Yaskawa INFORM job: A_ROOF_SIDE_0617_2_PAINT_0.JBI

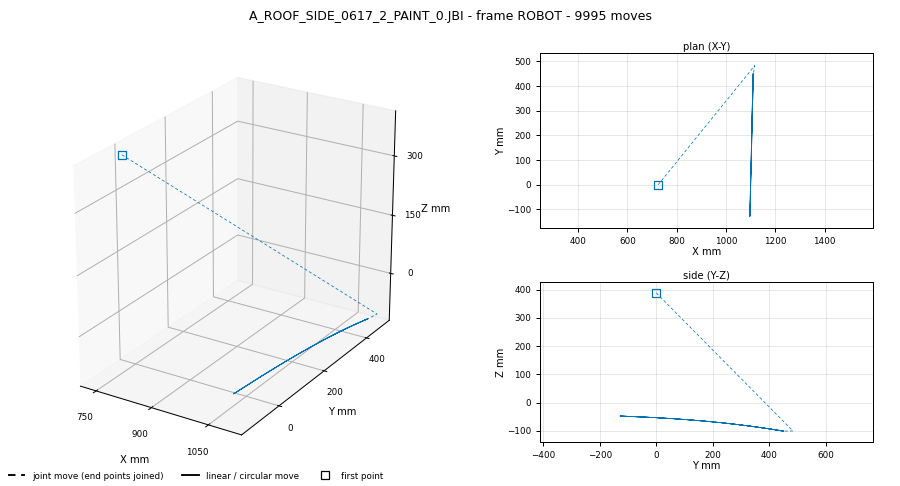
[picture p0: tool path of A_ROOF_SIDE_0617_2_PAINT_0.JBI in frame ROBOT, 9995 of 9995 moves have a stored position in this frame; points joined in program order, loops and branches not executed]
/JOB
//NAME A_ROOF_SIDE_0617_2_PAINT
//POS
///NPOS 9995,0,0,0,0,0
///TOOL 0
///USER 0
///POSTYPE ROBOT
///RECTAN
///RCONF 1,0,0,0,0,0,0,0,0,0,0,0,0,0,0,0,0,0,0,0,0,0,0,0
C00000=725.000,0.000,388.500,-180.000,-0.000,0.000
C00001=725.000,0.000,388.500,-180.000,-0.000,0.000
///TOOL 1
///USER 0
///POSTYPE ROBOT
///RECTAN
C00002=1116.924,483.635,-100.044,-178.124,16.519,151.125
C00003=1111.077,450.492,-100.420,-178.124,16.519,151.125
C00004=1111.072,450.245,-100.379,-178.121,16.509,151.122
C00005=1111.067,450.000,-100.338,-178.120,16.499,151.119
C00006=1111.061,449.753,-100.297,-178.118,16.490,151.116
C00007=1111.056,449.506,-100.255,-178.115,16.481,151.114
C00008=1111.050,449.260,-100.213,-178.113,16.472,151.111
C00009=1111.045,449.013,-100.173,-178.111,16.462,151.108
C00010=1111.039,448.767,-100.131,-178.109,16.453,151.105
C00011=1111.034,448.521,-100.090,-178.107,16.443,151.102
C00012=1111.028,448.275,-100.049,-178.105,16.434,151.099
C00013=1111.023,448.027,-100.007,-178.103,16.424,151.096
C00014=1111.017,447.781,-99.966,-178.102,16.415,151.094
C00015=1111.012,447.534,-99.925,-178.100,16.405,151.091
C00016=1111.007,447.289,-99.884,-178.099,16.395,151.088
C00017=1111.002,447.042,-99.843,-178.098,16.386,151.085
C00018=1110.996,446.796,-99.801,-178.096,16.376,151.082
C00019=1110.991,446.548,-99.760,-178.095,16.367,151.080
C00020=1110.985,446.302,-99.719,-178.093,16.357,151.077
C00021=1110.980,446.056,-99.678,-178.092,16.348,151.074
C00022=1110.975,445.810,-99.636,-178.092,16.338,151.072
C00023=1110.969,445.563,-99.595,-178.091,16.328,151.069
C00024=1110.963,445.317,-99.554,-178.090,16.318,151.066
C00025=1110.957,445.070,-99.513,-178.089,16.309,151.064
C00026=1110.952,444.824,-99.473,-178.089,16.299,151.061
C00027=1110.947,444.577,-99.431,-178.088,16.290,151.058
C00028=1110.941,444.330,-99.390,-178.088,16.280,151.056
C00029=1110.935,444.084,-99.349,-178.088,16.270,151.053
C00030=1110.930,443.838,-99.308,-178.088,16.260,151.051
C00031=1110.925,443.591,-99.267,-178.087,16.251,151.048
C00032=1110.919,443.345,-99.226,-178.087,16.241,151.046
C00033=1110.915,443.099,-99.185,-178.088,16.231,151.043
C00034=1110.909,442.852,-99.144,-178.088,16.221,151.041
C00035=1110.903,442.605,-99.103,-178.088,16.212,151.038
C00036=1110.898,442.359,-99.062,-178.089,16.202,151.036
C00037=1110.892,442.113,-99.022,-178.088,16.192,151.033
C00038=1110.887,441.866,-98.981,-178.089,16.182,151.031
C00039=1110.881,441.620,-98.940,-178.089,16.173,151.028
C00040=1110.876,441.373,-98.899,-178.089,16.164,151.026
C00041=1110.870,441.127,-98.858,-178.090,16.154,151.024
C00042=1110.864,440.880,-98.818,-178.090,16.145,151.021
C00043=1110.859,440.634,-98.777,-178.090,16.136,151.019
C00044=1110.853,440.387,-98.736,-178.091,16.126,151.017
C00045=1110.848,440.141,-98.695,-178.092,16.117,151.014
C00046=1110.843,439.894,-98.655,-178.092,16.107,151.012
C00047=1110.837,439.648,-98.614,-178.093,16.098,151.010
C00048=1110.831,439.401,-98.573,-178.093,16.089,151.007
C00049=1110.826,439.155,-98.533,-178.093,16.080,151.005
C00050=1110.820,438.908,-98.493,-178.094,16.071,151.003
C00051=1110.814,438.661,-98.452,-178.095,16.061,151.001
C00052=1110.809,438.428,-98.413,-178.095,16.052,150.998
C00053=1110.804,438.194,-98.375,-178.095,16.044,150.996
C00054=1110.799,437.961,-98.337,-178.096,16.036,150.994
C00055=1110.794,437.728,-98.298,-178.096,16.027,150.992
C00056=1110.788,437.494,-98.260,-178.097,16.019,150.990
C00057=1110.783,437.261,-98.221,-178.098,16.010,150.988
C00058=1110.778,437.027,-98.183,-178.098,16.002,150.986
C00059=1110.773,436.795,-98.145,-178.099,15.993,150.984
C00060=1110.767,436.548,-98.105,-178.100,15.985,150.982
C00061=1110.761,436.301,-98.064,-178.100,15.976,150.980
C00062=1110.756,436.055,-98.023,-178.101,15.967,150.978
C00063=1110.751,435.808,-97.983,-178.102,15.958,150.976
C00064=1110.745,435.562,-97.944,-178.103,15.949,150.973
C00065=1110.740,435.315,-97.903,-178.103,15.941,150.971
C00066=1110.734,435.068,-97.862,-178.104,15.932,150.969
C00067=1110.729,434.822,-97.822,-178.104,15.924,150.967
C00068=1110.723,434.575,-97.782,-178.105,15.915,150.965
C00069=1110.718,434.329,-97.742,-178.106,15.906,150.963
C00070=1110.712,434.082,-97.701,-178.107,15.898,150.961
C00071=1110.707,433.836,-97.661,-178.108,15.889,150.959
C00072=1110.701,433.589,-97.621,-178.109,15.881,150.957
C00073=1110.696,433.343,-97.581,-178.110,15.872,150.955
C00074=1110.690,433.096,-97.540,-178.111,15.864,150.953
C00075=1110.684,432.849,-97.501,-178.111,15.856,150.951
C00076=1110.679,432.602,-97.460,-178.112,15.847,150.949
C00077=1110.674,432.356,-97.420,-178.113,15.839,150.947
C00078=1110.668,432.109,-97.381,-178.114,15.831,150.945
C00079=1110.662,431.862,-97.340,-178.115,15.823,150.943
C00080=1110.657,431.616,-97.301,-178.116,15.815,150.942
C00081=1110.651,431.369,-97.260,-178.117,15.807,150.940
C00082=1110.646,431.123,-97.220,-178.118,15.798,150.938
C00083=1110.640,430.876,-97.180,-178.119,15.790,150.936
C00084=1110.635,430.630,-97.140,-178.120,15.782,150.934
C00085=1110.629,430.383,-97.100,-178.121,15.774,150.932
C00086=1110.623,430.136,-97.060,-178.122,15.766,150.930
C00087=1110.618,429.889,-97.021,-178.123,15.758,150.928
C00088=1110.612,429.642,-96.980,-178.124,15.750,150.927
C00089=1110.607,429.396,-96.941,-178.125,15.742,150.925
C00090=1110.602,429.149,-96.901,-178.126,15.734,150.923
C00091=1110.596,428.903,-96.861,-178.127,15.726,150.921
C00092=1110.590,428.655,-96.821,-178.128,15.719,150.919
C00093=1110.585,428.410,-96.781,-178.130,15.711,150.918
C00094=1110.579,428.162,-96.742,-178.131,15.703,150.916
C00095=1110.574,427.916,-96.702,-178.132,15.695,150.914
C00096=1110.567,427.669,-96.662,-178.133,15.687,150.912
C00097=1110.563,427.422,-96.622,-178.134,15.680,150.911
C00098=1110.557,427.175,-96.583,-178.135,15.672,150.909
C00099=1110.551,426.929,-96.544,-178.136,15.665,150.907
C00100=1110.546,426.682,-96.503,-178.138,15.657,150.906
C00101=1110.540,426.436,-96.464,-178.139,15.649,150.904
C00102=1110.534,426.188,-96.425,-178.140,15.642,150.902
C00103=1110.529,425.942,-96.385,-178.141,15.635,150.901
C00104=1110.523,425.696,-96.345,-178.142,15.627,150.899
C00105=1110.518,425.448,-96.305,-178.144,15.620,150.897
C00106=1110.513,425.202,-96.266,-178.145,15.612,150.896
C00107=1110.507,424.955,-96.227,-178.146,15.604,150.894
C00108=1110.502,424.737,-96.191,-178.148,15.598,150.893
C00109=1110.497,424.520,-96.157,-178.149,15.591,150.891
C00110=1110.492,424.301,-96.122,-178.150,15.585,150.890
C00111=1110.487,424.083,-96.087,-178.151,15.579,150.888
C00112=1110.483,423.866,-96.052,-178.152,15.572,150.887
C00113=1110.477,423.649,-96.018,-178.153,15.566,150.885
C00114=1110.472,423.430,-95.983,-178.154,15.560,150.884
C00115=1110.468,423.213,-95.948,-178.155,15.553,150.883
C00116=1110.462,422.966,-95.909,-178.157,15.546,150.881
C00117=1110.456,422.719,-95.870,-178.158,15.538,150.880
C00118=1110.451,422.472,-95.830,-178.160,15.531,150.878
C00119=1110.446,422.226,-95.791,-178.161,15.524,150.877
C00120=1110.440,421.979,-95.752,-178.163,15.517,150.875
C00121=1110.434,421.732,-95.712,-178.164,15.510,150.874
C00122=1110.429,421.486,-95.673,-178.165,15.503,150.872
C00123=1110.422,421.238,-95.634,-178.167,15.496,150.871
C00124=1110.417,420.992,-95.595,-178.169,15.489,150.869
C00125=1110.412,420.745,-95.556,-178.170,15.483,150.868
C00126=1110.407,420.497,-95.516,-178.171,15.475,150.866
C00127=1110.401,420.251,-95.477,-178.173,15.468,150.865
C00128=1110.395,420.004,-95.438,-178.174,15.462,150.863
C00129=1110.389,419.757,-95.399,-178.176,15.455,150.862
C00130=1110.384,419.511,-95.360,-178.177,15.448,150.860
C00131=1110.378,419.263,-95.321,-178.179,15.441,150.859
C00132=1110.373,419.017,-95.282,-178.181,15.434,150.858
C00133=1110.367,418.770,-95.243,-178.182,15.428,150.856
C00134=1110.361,418.523,-95.203,-178.184,15.421,150.855
C00135=1110.356,418.276,-95.165,-178.185,15.415,150.854
C00136=1110.351,418.030,-95.126,-178.187,15.408,150.852
C00137=1110.345,417.783,-95.087,-178.188,15.401,150.851
C00138=1110.339,417.536,-95.048,-178.190,15.394,150.850
C00139=1110.334,417.289,-95.009,-178.191,15.388,150.848
C00140=1110.328,417.042,-94.970,-178.193,15.381,150.847
C00141=1110.323,416.795,-94.931,-178.194,15.375,150.845
C00142=1110.317,416.549,-94.892,-178.196,15.368,150.844
C00143=1110.311,416.301,-94.854,-178.197,15.362,150.843
C00144=1110.306,416.054,-94.814,-178.199,15.355,150.842
C00145=1110.301,415.807,-94.776,-178.201,15.349,150.840
C00146=1110.295,415.560,-94.737,-178.203,15.342,150.839
C00147=1110.288,415.314,-94.698,-178.204,15.336,150.838
C00148=1110.283,415.067,-94.660,-178.206,15.330,150.836
C00149=1110.277,414.820,-94.620,-178.208,15.323,150.835
C00150=1110.272,414.573,-94.582,-178.210,15.317,150.834
C00151=1110.267,414.326,-94.544,-178.211,15.311,150.833
C00152=1110.261,414.079,-94.505,-178.213,15.305,150.832
C00153=1110.255,413.832,-94.467,-178.215,15.298,150.830
C00154=1110.249,413.585,-94.427,-178.216,15.292,150.829
C00155=1110.244,413.338,-94.389,-178.218,15.286,150.828
C00156=1110.238,413.091,-94.350,-178.220,15.280,150.827
C00157=1110.232,412.844,-94.312,-178.222,15.274,150.826
C00158=1110.227,412.597,-94.274,-178.224,15.267,150.824
C00159=1110.222,412.351,-94.235,-178.225,15.261,150.823
C00160=1110.216,412.103,-94.196,-178.227,15.255,150.822
C00161=1110.211,411.856,-94.157,-178.229,15.249,150.821
C00162=1110.205,411.609,-94.120,-178.231,15.243,150.820
C00163=1110.199,411.363,-94.081,-178.232,15.237,150.818
C00164=1110.194,411.151,-94.048,-178.234,15.232,150.818
C00165=1110.190,410.939,-94.015,-178.235,15.227,150.817
C00166=1110.185,410.729,-93.982,-178.237,15.222,150.816
C00167=1110.180,410.517,-93.949,-178.238,15.217,150.815
C00168=1110.176,410.305,-93.917,-178.240,15.211,150.814
C00169=1110.171,410.094,-93.883,-178.241,15.207,150.813
C00170=1110.166,409.883,-93.851,-178.243,15.201,150.812
C00171=1110.161,409.671,-93.818,-178.244,15.197,150.811
C00172=1110.156,409.424,-93.780,-178.247,15.190,150.810
C00173=1110.150,409.177,-93.740,-178.248,15.185,150.809
C00174=1110.144,408.931,-93.703,-178.250,15.179,150.808
C00175=1110.139,408.683,-93.664,-178.252,15.173,150.806
C00176=1110.134,408.436,-93.626,-178.253,15.168,150.805
C00177=1110.128,408.190,-93.588,-178.256,15.161,150.804
C00178=1110.123,407.943,-93.550,-178.258,15.156,150.803
C00179=1110.116,407.695,-93.512,-178.259,15.150,150.802
C00180=1110.111,407.448,-93.473,-178.261,15.145,150.801
C00181=1110.105,407.201,-93.436,-178.263,15.139,150.800
C00182=1110.100,406.954,-93.397,-178.266,15.133,150.799
C00183=1110.095,406.707,-93.359,-178.267,15.127,150.798
C00184=1110.089,406.461,-93.321,-178.269,15.122,150.797
C00185=1110.084,406.213,-93.283,-178.271,15.116,150.796
C00186=1110.077,405.966,-93.245,-178.273,15.111,150.795
C00187=1110.072,405.719,-93.206,-178.275,15.105,150.794
C00188=1110.066,405.472,-93.169,-178.277,15.100,150.793
C00189=1110.061,405.225,-93.130,-178.279,15.095,150.792
C00190=1110.055,404.978,-93.093,-178.281,15.089,150.791
C00191=1110.049,404.731,-93.056,-178.283,15.084,150.791
C00192=1110.044,404.484,-93.017,-178.285,15.078,150.790
C00193=1110.038,404.237,-92.979,-178.287,15.073,150.789
C00194=1110.033,403.989,-92.941,-178.289,15.067,150.788
C00195=1110.027,403.743,-92.903,-178.291,15.062,150.787
C00196=1110.021,403.496,-92.865,-178.293,15.057,150.786
C00197=1110.016,403.248,-92.828,-178.295,15.051,150.785
C00198=1110.010,403.002,-92.790,-178.297,15.046,150.784
C00199=1110.004,402.755,-92.752,-178.299,15.041,150.783
C00200=1109.999,402.508,-92.714,-178.301,15.035,150.782
C00201=1109.993,402.260,-92.677,-178.303,15.030,150.781
C00202=1109.987,402.014,-92.639,-178.305,15.025,150.781
C00203=1109.982,401.767,-92.601,-178.307,15.020,150.780
C00204=1109.977,401.519,-92.563,-178.309,15.014,150.779
C00205=1109.971,401.273,-92.526,-178.312,15.009,150.778
C00206=1109.966,401.025,-92.487,-178.313,15.004,150.777
C00207=1109.960,400.778,-92.450,-178.316,14.999,150.776
C00208=1109.954,400.531,-92.413,-178.317,14.995,150.775
C00209=1109.949,400.284,-92.375,-178.319,14.989,150.775
C00210=1109.943,400.037,-92.337,-178.321,14.984,150.774
C00211=1109.937,399.790,-92.299,-178.324,14.979,150.773
C00212=1109.932,399.543,-92.262,-178.326,14.974,150.772
C00213=1109.926,399.296,-92.225,-178.328,14.969,150.771
C00214=1109.921,399.048,-92.187,-178.330,14.964,150.771
C00215=1109.915,398.801,-92.149,-178.332,14.959,150.770
C00216=1109.909,398.554,-92.112,-178.335,14.954,150.769
C00217=1109.904,398.308,-92.074,-178.337,14.949,150.768
C00218=1109.898,398.060,-92.037,-178.339,14.945,150.767
C00219=1109.892,397.813,-92.000,-178.341,14.940,150.767
C00220=1109.888,397.601,-91.967,-178.343,14.936,150.766
C00221=1109.883,397.390,-91.935,-178.345,14.931,150.765
C00222=1109.878,397.178,-91.904,-178.347,14.927,150.765
C00223=1109.873,396.966,-91.871,-178.349,14.923,150.764
C00224=1109.868,396.755,-91.839,-178.350,14.919,150.763
C00225=1109.863,396.543,-91.808,-178.352,14.915,150.763
C00226=1109.858,396.331,-91.775,-178.354,14.911,150.762
C00227=1109.854,396.119,-91.743,-178.356,14.907,150.762
C00228=1109.848,395.872,-91.706,-178.358,14.902,150.761
C00229=1109.842,395.625,-91.669,-178.360,14.897,150.760
C00230=1109.837,395.378,-91.632,-178.363,14.892,150.760
C00231=1109.831,395.132,-91.594,-178.365,14.887,150.759
C00232=1109.826,394.884,-91.557,-178.367,14.883,150.758
C00233=1109.820,394.637,-91.520,-178.369,14.878,150.757
C00234=1109.815,394.389,-91.483,-178.372,14.874,150.757
C00235=1109.809,394.143,-91.445,-178.374,14.869,150.756
C00236=1109.803,393.895,-91.408,-178.376,14.865,150.755
C00237=1109.797,393.648,-91.371,-178.379,14.860,150.755
C00238=1109.792,393.401,-91.334,-178.381,14.855,150.754
C00239=1109.787,393.155,-91.297,-178.383,14.850,150.753
C00240=1109.781,392.907,-91.260,-178.385,14.847,150.753
C00241=1109.775,392.660,-91.223,-178.387,14.842,150.752
C00242=1109.770,392.413,-91.186,-178.390,14.837,150.752
C00243=1109.764,392.165,-91.149,-178.393,14.832,150.751
C00244=1109.758,391.918,-91.112,-178.394,14.828,150.750
C00245=1109.752,391.671,-91.074,-178.397,14.824,150.750
C00246=1109.746,391.424,-91.037,-178.400,14.819,150.749
C00247=1109.741,391.177,-91.001,-178.401,14.815,150.749
C00248=1109.736,390.930,-90.964,-178.404,14.811,150.748
C00249=1109.729,390.683,-90.927,-178.407,14.806,150.748
C00250=1109.724,390.436,-90.890,-178.410,14.802,150.747
C00251=1109.718,390.188,-90.853,-178.411,14.798,150.746
C00252=1109.713,389.942,-90.816,-178.414,14.793,150.746
C00253=1109.707,389.694,-90.780,-178.417,14.788,150.745
C00254=1109.701,389.447,-90.743,-178.419,14.785,150.745
C00255=1109.696,389.200,-90.706,-178.421,14.780,150.744
C00256=1109.690,388.952,-90.669,-178.424,14.776,150.744
C00257=1109.684,388.706,-90.633,-178.426,14.772,150.743
C00258=1109.679,388.459,-90.596,-178.429,14.767,150.743
C00259=1109.673,388.211,-90.559,-178.432,14.763,150.742
C00260=1109.667,387.964,-90.522,-178.433,14.759,150.741
C00261=1109.662,387.718,-90.486,-178.436,14.755,150.741
C00262=1109.656,387.470,-90.449,-178.438,14.751,150.740
C00263=1109.650,387.223,-90.412,-178.441,14.747,150.740
C00264=1109.645,386.976,-90.376,-178.444,14.742,150.739
C00265=1109.640,386.729,-90.339,-178.446,14.738,150.739
C00266=1109.633,386.481,-90.303,-178.448,14.734,150.738
C00267=1109.628,386.234,-90.266,-178.451,14.729,150.738
C00268=1109.623,385.987,-90.229,-178.453,14.726,150.738
C00269=1109.617,385.740,-90.193,-178.456,14.721,150.737
C00270=1109.611,385.492,-90.156,-178.458,14.718,150.737
C00271=1109.606,385.246,-90.120,-178.461,14.713,150.736
C00272=1109.600,384.999,-90.083,-178.464,14.709,150.736
C00273=1109.594,384.751,-90.047,-178.466,14.706,150.735
C00274=1109.589,384.504,-90.011,-178.469,14.701,150.735
C00275=1109.583,384.257,-89.974,-178.471,14.697,150.734
C00276=1109.573,383.845,-89.913,-178.476,14.691,150.734
C00277=1109.564,383.434,-89.853,-178.479,14.684,150.733
C00278=1109.555,383.023,-89.792,-178.484,14.677,150.732
C00279=1109.546,382.612,-89.732,-178.488,14.671,150.732
C00280=1109.540,382.364,-89.695,-178.491,14.667,150.731
C00281=1109.534,382.117,-89.659,-178.493,14.663,150.731
C00282=1109.529,381.870,-89.623,-178.496,14.660,150.730
C00283=1109.523,381.622,-89.587,-178.498,14.656,150.730
C00284=1109.517,381.375,-89.550,-178.501,14.652,150.730
C00285=1109.512,381.128,-89.514,-178.504,14.649,150.729
C00286=1109.506,380.881,-89.478,-178.507,14.644,150.729
C00287=1109.500,380.633,-89.442,-178.509,14.641,150.728
C00288=1109.495,380.386,-89.405,-178.512,14.637,150.728
C00289=1109.489,380.139,-89.370,-178.514,14.633,150.728
C00290=1109.483,379.891,-89.333,-178.517,14.629,150.728
C00291=1109.478,379.644,-89.297,-178.520,14.626,150.727
C00292=1109.472,379.397,-89.261,-178.523,14.622,150.727
C00293=1109.467,379.150,-89.225,-178.525,14.618,150.726
C00294=1109.461,378.902,-89.189,-178.528,14.614,150.726
C00295=1109.455,378.656,-89.153,-178.530,14.611,150.726
C00296=1109.450,378.408,-89.117,-178.533,14.608,150.726
C00297=1109.444,378.160,-89.081,-178.536,14.604,150.725
C00298=1109.438,377.914,-89.045,-178.538,14.600,150.725
C00299=1109.433,377.666,-89.009,-178.542,14.596,150.725
C00300=1109.427,377.419,-88.973,-178.544,14.593,150.724
C00301=1109.421,377.171,-88.937,-178.547,14.589,150.724
C00302=1109.416,376.925,-88.901,-178.549,14.585,150.724
C00303=1109.410,376.677,-88.865,-178.552,14.582,150.723
C00304=1109.405,376.430,-88.830,-178.555,14.578,150.723
C00305=1109.399,376.182,-88.794,-178.557,14.575,150.723
C00306=1109.393,375.936,-88.758,-178.561,14.571,150.723
C00307=1109.388,375.688,-88.722,-178.563,14.568,150.722
C00308=1109.382,375.441,-88.686,-178.566,14.564,150.722
C00309=1109.376,375.194,-88.650,-178.569,14.561,150.722
C00310=1109.371,374.947,-88.615,-178.571,14.557,150.722
C00311=1109.366,374.699,-88.579,-178.574,14.554,150.721
C00312=1109.360,374.452,-88.543,-178.577,14.550,150.721
C00313=1109.354,374.205,-88.507,-178.580,14.547,150.721
C00314=1109.348,373.957,-88.471,-178.583,14.543,150.721
C00315=1109.342,373.710,-88.436,-178.585,14.540,150.720
C00316=1109.336,373.462,-88.400,-178.588,14.537,150.720
C00317=1109.331,373.215,-88.365,-178.591,14.533,150.720
C00318=1109.325,372.968,-88.329,-178.594,14.530,150.720
C00319=1109.319,372.721,-88.294,-178.596,14.527,150.719
C00320=1109.314,372.473,-88.257,-178.599,14.524,150.719
C00321=1109.309,372.226,-88.222,-178.602,14.520,150.719
C00322=1109.303,371.978,-88.186,-178.605,14.517,150.719
C00323=1109.297,371.731,-88.151,-178.608,14.514,150.719
C00324=1109.291,371.483,-88.115,-178.611,14.510,150.719
C00325=1109.286,371.236,-88.080,-178.614,14.507,150.718
C00326=1109.280,370.989,-88.044,-178.616,14.504,150.718
C00327=1109.274,370.742,-88.009,-178.620,14.500,150.718
C00328=1109.266,370.357,-87.954,-178.624,14.495,150.718
C00329=1109.256,369.972,-87.899,-178.628,14.491,150.718
C00330=1109.248,369.587,-87.844,-178.633,14.485,150.717
C00331=1109.240,369.202,-87.789,-178.637,14.481,150.717
C00332=1109.233,368.955,-87.753,-178.640,14.478,150.717
C00333=1109.228,368.708,-87.718,-178.643,14.474,150.717
C00334=1109.222,368.459,-87.683,-178.646,14.471,150.717
C00335=1109.217,368.212,-87.648,-178.649,14.468,150.717
C00336=1109.211,367.966,-87.612,-178.651,14.465,150.716
C00337=1109.206,367.717,-87.577,-178.655,14.461,150.716
C00338=1109.200,367.471,-87.542,-178.658,14.459,150.716
C00339=1109.194,367.224,-87.507,-178.661,14.456,150.716
C00340=1109.188,366.975,-87.472,-178.663,14.453,150.716
C00341=1109.183,366.728,-87.437,-178.667,14.449,150.716
C00342=1109.177,366.481,-87.401,-178.669,14.446,150.716
C00343=1109.172,366.233,-87.366,-178.672,14.443,150.716
C00344=1109.166,365.986,-87.331,-178.675,14.441,150.716
C00345=1109.160,365.738,-87.295,-178.678,14.438,150.716
C00346=1109.155,365.491,-87.261,-178.681,14.434,150.715
C00347=1109.149,365.244,-87.226,-178.684,14.431,150.715
C00348=1109.143,364.996,-87.191,-178.687,14.428,150.715
C00349=1109.138,364.749,-87.155,-178.690,14.426,150.715
C00350=1109.132,364.501,-87.120,-178.693,14.423,150.715
C00351=1109.126,364.254,-87.086,-178.696,14.419,150.715
C00352=1109.121,364.006,-87.051,-178.699,14.416,150.715
C00353=1109.115,363.759,-87.015,-178.702,14.414,150.715
C00354=1109.110,363.511,-86.981,-178.705,14.411,150.715
C00355=1109.104,363.264,-86.946,-178.708,14.408,150.715
C00356=1109.098,363.016,-86.911,-178.711,14.405,150.715
C00357=1109.092,362.769,-86.875,-178.714,14.402,150.715
C00358=1109.087,362.522,-86.841,-178.717,14.399,150.715
C00359=1109.081,362.274,-86.807,-178.720,14.396,150.715
C00360=1109.075,362.027,-86.771,-178.723,14.393,150.715
C00361=1109.070,361.779,-86.737,-178.726,14.391,150.715
C00362=1109.064,361.532,-86.702,-178.729,14.388,150.715
C00363=1109.058,361.284,-86.667,-178.732,14.385,150.715
C00364=1109.053,361.037,-86.633,-178.736,14.382,150.715
C00365=1109.047,360.789,-86.598,-178.739,14.379,150.715
C00366=1109.041,360.541,-86.562,-178.741,14.376,150.715
C00367=1109.036,360.294,-86.528,-178.745,14.374,150.715
C00368=1109.030,360.047,-86.493,-178.747,14.371,150.715
C00369=1109.024,359.800,-86.459,-178.751,14.369,150.715
C00370=1109.019,359.552,-86.424,-178.753,14.366,150.715
C00371=1109.013,359.304,-86.390,-178.757,14.363,150.715
C00372=1109.008,359.057,-86.355,-178.759,14.361,150.715
C00373=1109.002,358.809,-86.320,-178.763,14.358,150.715
C00374=1108.996,358.562,-86.285,-178.767,14.355,150.715
C00375=1108.991,358.314,-86.251,-178.769,14.352,150.715
C00376=1108.985,358.067,-86.216,-178.773,14.350,150.715
C00377=1108.980,357.819,-86.182,-178.775,14.347,150.715
C00378=1108.973,357.571,-86.147,-178.779,14.344,150.715
C00379=1108.968,357.324,-86.113,-178.782,14.342,150.715
C00380=1108.959,356.954,-86.061,-178.786,14.338,150.715
C00381=1108.950,356.584,-86.010,-178.791,14.334,150.715
C00382=1108.942,356.214,-85.958,-178.796,14.330,150.715
C00383=1108.934,355.844,-85.907,-178.800,14.326,150.715
C00384=1108.928,355.596,-85.872,-178.803,14.324,150.716
C00385=1108.922,355.348,-85.838,-178.806,14.322,150.716
C00386=1108.917,355.101,-85.804,-178.810,14.319,150.716
C00387=1108.911,354.854,-85.770,-178.813,14.317,150.716
C00388=1108.906,354.606,-85.735,-178.816,14.314,150.716
C00389=1108.900,354.358,-85.701,-178.819,14.311,150.716
C00390=1108.894,354.110,-85.666,-178.822,14.309,150.716
C00391=1108.889,353.863,-85.632,-178.825,14.306,150.716
C00392=1108.883,353.616,-85.598,-178.828,14.304,150.716
C00393=1108.878,353.368,-85.564,-178.832,14.302,150.716
C00394=1108.872,353.120,-85.530,-178.835,14.299,150.716
C00395=1108.866,352.873,-85.496,-178.838,14.297,150.717
C00396=1108.860,352.625,-85.461,-178.841,14.294,150.717
C00397=1108.855,352.377,-85.427,-178.844,14.292,150.717
C00398=1108.849,352.130,-85.393,-178.848,14.290,150.717
C00399=1108.843,351.882,-85.359,-178.851,14.287,150.717
C00400=1108.838,351.635,-85.325,-178.854,14.285,150.717
C00401=1108.832,351.387,-85.291,-178.857,14.282,150.717
C00402=1108.826,351.140,-85.257,-178.861,14.280,150.718
C00403=1108.820,350.892,-85.223,-178.864,14.277,150.718
C00404=1108.815,350.644,-85.188,-178.867,14.275,150.718
C00405=1108.809,350.397,-85.154,-178.870,14.273,150.718
C00406=1108.804,350.149,-85.121,-178.874,14.270,150.718
C00407=1108.798,349.901,-85.087,-178.877,14.268,150.718
C00408=1108.792,349.654,-85.053,-178.880,14.266,150.719
C00409=1108.787,349.406,-85.019,-178.883,14.263,150.719
C00410=1108.781,349.159,-84.985,-178.887,14.261,150.719
C00411=1108.775,348.911,-84.951,-178.890,14.259,150.719
C00412=1108.770,348.664,-84.917,-178.893,14.256,150.719
C00413=1108.763,348.416,-84.883,-178.897,14.254,150.719
C00414=1108.758,348.168,-84.850,-178.900,14.252,150.720
C00415=1108.753,347.920,-84.815,-178.903,14.249,150.720
C00416=1108.747,347.673,-84.781,-178.906,14.248,150.720
C00417=1108.741,347.425,-84.748,-178.909,14.246,150.720
C00418=1108.735,347.178,-84.713,-178.912,14.243,150.720
C00419=1108.730,346.930,-84.680,-178.916,14.241,150.720
C00420=1108.724,346.682,-84.646,-178.919,14.239,150.721
C00421=1108.718,346.434,-84.613,-178.923,14.237,150.721
C00422=1108.713,346.187,-84.579,-178.926,14.234,150.721
C00423=1108.707,345.939,-84.545,-178.929,14.232,150.721
C00424=1108.701,345.691,-84.512,-178.932,14.230,150.721
C00425=1108.696,345.444,-84.477,-178.936,14.228,150.722
C00426=1108.691,345.196,-84.444,-178.939,14.226,150.722
C00427=1108.685,344.949,-84.410,-178.942,14.224,150.722
C00428=1108.679,344.701,-84.377,-178.946,14.222,150.722
C00429=1108.673,344.453,-84.344,-178.949,14.220,150.723
C00430=1108.667,344.206,-84.310,-178.952,14.217,150.723
C00431=1108.662,343.958,-84.277,-178.956,14.215,150.723
C00432=1108.654,343.590,-84.227,-178.961,14.212,150.724
C00433=1108.645,343.223,-84.177,-178.965,14.209,150.724
C00434=1108.636,342.854,-84.127,-178.971,14.206,150.724
C00435=1108.628,342.486,-84.077,-178.976,14.203,150.725
C00436=1108.622,342.238,-84.044,-178.978,14.201,150.725
C00437=1108.616,341.991,-84.010,-178.982,14.199,150.725
C00438=1108.611,341.743,-83.977,-178.985,14.197,150.725
C00439=1108.605,341.495,-83.944,-178.989,14.195,150.726
C00440=1108.600,341.247,-83.910,-178.992,14.193,150.726
C00441=1108.594,340.999,-83.877,-178.996,14.191,150.726
C00442=1108.589,340.751,-83.844,-178.999,14.189,150.727
C00443=1108.583,340.505,-83.810,-179.002,14.187,150.727
C00444=1108.577,340.257,-83.777,-179.006,14.185,150.727
C00445=1108.571,340.009,-83.744,-179.009,14.183,150.727
C00446=1108.566,339.761,-83.710,-179.012,14.181,150.728
C00447=1108.560,339.513,-83.677,-179.015,14.179,150.728
C00448=1108.555,339.265,-83.644,-179.019,14.177,150.728
C00449=1108.549,339.017,-83.610,-179.022,14.175,150.728
C00450=1108.543,338.770,-83.578,-179.026,14.173,150.729
C00451=1108.537,338.522,-83.544,-179.029,14.171,150.729
C00452=1108.532,338.274,-83.511,-179.032,14.170,150.729
C00453=1108.527,338.027,-83.478,-179.036,14.168,150.730
C00454=1108.521,337.779,-83.445,-179.040,14.166,150.730
C00455=1108.515,337.531,-83.412,-179.043,14.164,150.730
C00456=1108.509,337.283,-83.379,-179.046,14.163,150.731
C00457=1108.503,337.036,-83.346,-179.049,14.161,150.731
C00458=1108.498,336.788,-83.313,-179.053,14.159,150.731
C00459=1108.492,336.540,-83.279,-179.057,14.157,150.732
C00460=1108.486,336.292,-83.246,-179.060,14.155,150.732
C00461=1108.481,336.045,-83.214,-179.063,14.153,150.732
C00462=1108.476,335.797,-83.181,-179.067,14.151,150.733
C00463=1108.469,335.549,-83.148,-179.071,14.150,150.733
C00464=1108.464,335.301,-83.115,-179.073,14.148,150.733
C00465=1108.458,335.053,-83.081,-179.077,14.146,150.734
C00466=1108.452,334.806,-83.049,-179.080,14.144,150.734
C00467=1108.447,334.558,-83.016,-179.084,14.142,150.734
C00468=1108.441,334.310,-82.984,-179.087,14.141,150.735
C00469=1108.435,334.062,-82.950,-179.091,14.139,150.735
C00470=1108.430,333.814,-82.917,-179.094,14.137,150.736
C00471=1108.423,333.567,-82.884,-179.098,14.135,150.736
C00472=1108.419,333.319,-82.852,-179.101,14.134,150.736
C00473=1108.413,333.071,-82.819,-179.105,14.132,150.737
C00474=1108.407,332.824,-82.786,-179.108,14.130,150.737
C00475=1108.402,332.575,-82.753,-179.111,14.129,150.737
C00476=1108.395,332.327,-82.721,-179.115,14.127,150.738
C00477=1108.391,332.080,-82.688,-179.119,14.126,150.738
C00478=1108.385,331.832,-82.656,-179.122,14.124,150.738
C00479=1108.378,331.584,-82.623,-179.125,14.122,150.739
C00480=1108.373,331.337,-82.590,-179.129,14.120,150.739
C00481=1108.367,331.088,-82.558,-179.132,14.119,150.740
C00482=1108.361,330.841,-82.525,-179.136,14.118,150.740
C00483=1108.356,330.593,-82.493,-179.139,14.116,150.740
C00484=1108.347,330.219,-82.442,-179.144,14.114,150.741
C00485=1108.338,329.845,-82.394,-179.150,14.111,150.742
C00486=1108.329,329.471,-82.344,-179.155,14.109,150.742
C00487=1108.321,329.097,-82.295,-179.161,14.106,150.743
C00488=1108.315,328.849,-82.263,-179.164,14.105,150.743
C00489=1108.309,328.601,-82.231,-179.168,14.104,150.744
C00490=1108.304,328.353,-82.198,-179.171,14.102,150.744
C00491=1108.298,328.105,-82.166,-179.174,14.101,150.745
C00492=1108.292,327.857,-82.133,-179.178,14.099,150.745
C00493=1108.286,327.609,-82.101,-179.182,14.097,150.746
C00494=1108.281,327.362,-82.069,-179.185,14.096,150.746
C00495=1108.275,327.114,-82.036,-179.189,14.094,150.746
C00496=1108.269,326.865,-82.004,-179.192,14.093,150.747
C00497=1108.264,326.618,-81.971,-179.196,14.092,150.747
C00498=1108.258,326.370,-81.939,-179.200,14.090,150.748
C00499=1108.252,326.122,-81.907,-179.202,14.089,150.748
C00500=1108.246,325.875,-81.875,-179.206,14.087,150.749
C00501=1108.241,325.626,-81.842,-179.210,14.085,150.749
C00502=1108.235,325.378,-81.810,-179.213,14.084,150.750
C00503=1108.229,325.131,-81.778,-179.217,14.083,150.750
C00504=1108.223,324.883,-81.746,-179.220,14.082,150.751
C00505=1108.218,324.635,-81.713,-179.224,14.080,150.751
C00506=1108.213,324.387,-81.682,-179.228,14.078,150.751
C00507=1108.206,324.140,-81.649,-179.231,14.077,150.752
C00508=1108.200,323.891,-81.617,-179.235,14.075,150.752
C00509=1108.195,323.644,-81.585,-179.238,14.074,150.753
C00510=1108.189,323.396,-81.553,-179.242,14.073,150.753
C00511=1108.184,323.148,-81.521,-179.245,14.072,150.754
C00512=1108.178,322.900,-81.488,-179.249,14.070,150.754
C00513=1108.172,322.652,-81.456,-179.253,14.068,150.755
C00514=1108.167,322.404,-81.425,-179.256,14.067,150.755
C00515=1108.161,322.156,-81.393,-179.260,14.066,150.756
C00516=1108.155,321.909,-81.361,-179.263,14.065,150.756
C00517=1108.150,321.660,-81.328,-179.267,14.063,150.757
C00518=1108.145,321.413,-81.297,-179.270,14.062,150.757
C00519=1108.139,321.164,-81.265,-179.274,14.060,150.758
C00520=1108.133,320.917,-81.233,-179.278,14.059,150.758
C00521=1108.127,320.669,-81.201,-179.281,14.058,150.759
C00522=1108.122,320.421,-81.169,-179.285,14.056,150.759
C00523=1108.116,320.173,-81.137,-179.288,14.055,150.759
C00524=1108.111,319.925,-81.106,-179.292,14.054,150.760
C00525=1108.105,319.677,-81.074,-179.295,14.053,150.760
C00526=1108.099,319.430,-81.042,-179.299,14.051,150.761
C00527=1108.093,319.182,-81.010,-179.302,14.050,150.762
C00528=1108.088,318.934,-80.978,-179.306,14.049,150.762
C00529=1108.082,318.686,-80.946,-179.309,14.048,150.763
C00530=1108.077,318.438,-80.914,-179.313,14.046,150.763
C00531=1108.071,318.190,-80.882,-179.316,14.045,150.764
C00532=1108.066,317.942,-80.850,-179.320,14.043,150.764
C00533=1108.060,317.694,-80.818,-179.324,14.042,150.765
C00534=1108.055,317.446,-80.787,-179.328,14.041,150.765
C00535=1108.049,317.198,-80.755,-179.332,14.040,150.766
C00536=1108.040,316.817,-80.706,-179.337,14.038,150.766
C00537=1108.031,316.436,-80.658,-179.342,14.036,150.767
C00538=1108.023,316.055,-80.610,-179.348,14.034,150.768
C00539=1108.014,315.673,-80.561,-179.353,14.032,150.769
C00540=1108.009,315.426,-80.529,-179.357,14.031,150.769
C00541=1108.003,315.178,-80.497,-179.360,14.030,150.770
C00542=1107.997,314.930,-80.466,-179.364,14.028,150.770
C00543=1107.992,314.681,-80.434,-179.368,14.028,150.771
C00544=1107.985,314.434,-80.403,-179.372,14.026,150.772
C00545=1107.980,314.187,-80.372,-179.375,14.025,150.772
C00546=1107.974,313.938,-80.340,-179.378,14.025,150.773
C00547=1107.968,313.690,-80.309,-179.383,14.023,150.773
C00548=1107.962,313.442,-80.277,-179.386,14.022,150.774
C00549=1107.957,313.194,-80.246,-179.390,14.021,150.774
C00550=1107.951,312.946,-80.214,-179.393,14.020,150.775
C00551=1107.945,312.699,-80.183,-179.397,14.019,150.776
C00552=1107.939,312.450,-80.152,-179.401,14.018,150.776
C00553=1107.934,312.202,-80.120,-179.405,14.017,150.777
C00554=1107.928,311.955,-80.090,-179.408,14.016,150.777
C00555=1107.922,311.706,-80.058,-179.412,14.014,150.778
C00556=1107.917,311.459,-80.026,-179.416,14.014,150.779
C00557=1107.911,311.211,-79.996,-179.419,14.013,150.779
C00558=1107.905,310.963,-79.964,-179.423,14.012,150.780
C00559=1107.900,310.715,-79.933,-179.427,14.011,150.780
C00560=1107.893,310.467,-79.902,-179.430,14.009,150.781
C00561=1107.888,310.219,-79.871,-179.434,14.009,150.782
C00562=1107.882,309.971,-79.840,-179.438,14.007,150.782
C00563=1107.876,309.723,-79.808,-179.441,14.007,150.783
C00564=1107.871,309.475,-79.777,-179.446,14.005,150.783
C00565=1107.865,309.227,-79.746,-179.449,14.004,150.784
C00566=1107.859,308.978,-79.715,-179.452,14.004,150.785
C00567=1107.853,308.731,-79.684,-179.456,14.003,150.785
C00568=1107.848,308.483,-79.653,-179.460,14.002,150.786
C00569=1107.842,308.236,-79.622,-179.464,14.000,150.786
C00570=1107.836,307.987,-79.591,-179.467,14.000,150.787
C00571=1107.831,307.739,-79.560,-179.472,13.999,150.788
C00572=1107.825,307.492,-79.528,-179.475,13.998,150.788
C00573=1107.820,307.243,-79.497,-179.478,13.997,150.789
C00574=1107.814,306.995,-79.467,-179.483,13.996,150.789
C00575=1107.808,306.748,-79.435,-179.486,13.995,150.790
C00576=1107.803,306.500,-79.405,-179.490,13.994,150.791
C00577=1107.797,306.251,-79.374,-179.493,13.993,150.791
C00578=1107.791,306.003,-79.343,-179.498,13.992,150.792
C00579=1107.786,305.756,-79.311,-179.501,13.991,150.792
C00580=1107.780,305.508,-79.281,-179.504,13.990,150.793
C00581=1107.775,305.260,-79.250,-179.509,13.989,150.794
C00582=1107.768,305.011,-79.219,-179.512,13.989,150.794
C00583=1107.763,304.763,-79.189,-179.516,13.987,150.795
C00584=1107.757,304.516,-79.157,-179.519,13.986,150.796
C00585=1107.751,304.268,-79.127,-179.523,13.986,150.796
C00586=1107.746,304.020,-79.096,-179.527,13.985,150.797
C00587=1107.740,303.772,-79.066,-179.531,13.984,150.798
C00588=1107.732,303.394,-79.019,-179.536,13.983,150.799
C00589=1107.723,303.014,-78.972,-179.543,13.981,150.800
C00590=1107.714,302.636,-78.925,-179.548,13.979,150.800
C00591=1107.705,302.257,-78.878,-179.554,13.978,150.801
C00592=1107.700,302.009,-78.847,-179.557,13.978,150.802
C00593=1107.694,301.762,-78.817,-179.561,13.976,150.803
C00594=1107.689,301.513,-78.786,-179.565,13.976,150.803
C00595=1107.683,301.266,-78.755,-179.568,13.975,150.804
C00596=1107.678,301.018,-78.725,-179.573,13.974,150.805
C00597=1107.673,300.770,-78.694,-179.576,13.974,150.806
C00598=1107.667,300.521,-78.664,-179.580,13.972,150.806
C00599=1107.661,300.273,-78.634,-179.584,13.972,150.807
C00600=1107.655,300.025,-78.603,-179.587,13.971,150.807
C00601=1107.650,299.777,-78.572,-179.591,13.970,150.808
C00602=1107.644,299.529,-78.542,-179.595,13.969,150.809
C00603=1107.639,299.281,-78.511,-179.598,13.969,150.809
C00604=1107.633,299.033,-78.481,-179.603,13.967,150.810
C00605=1107.627,298.785,-78.450,-179.606,13.967,150.811
C00606=1107.621,298.537,-78.420,-179.610,13.966,150.811
C00607=1107.617,298.289,-78.390,-179.614,13.965,150.812
C00608=1107.611,298.041,-78.359,-179.617,13.964,150.813
C00609=1107.605,297.793,-78.329,-179.621,13.964,150.813
C00610=1107.599,297.545,-78.299,-179.625,13.963,150.814
C00611=1107.593,297.297,-78.268,-179.629,13.963,150.815
C00612=1107.588,297.049,-78.239,-179.632,13.962,150.816
C00613=1107.583,296.801,-78.208,-179.637,13.961,150.816
C00614=1107.577,296.553,-78.177,-179.640,13.960,150.817
C00615=1107.571,296.305,-78.147,-179.644,13.960,150.818
C00616=1107.565,296.056,-78.117,-179.648,13.959,150.818
C00617=1107.559,295.808,-78.087,-179.652,13.958,150.819
C00618=1107.553,295.560,-78.056,-179.655,13.958,150.820
C00619=1107.548,295.312,-78.027,-179.660,13.957,150.820
C00620=1107.542,295.064,-77.996,-179.663,13.956,150.821
C00621=1107.536,294.816,-77.966,-179.667,13.956,150.822
C00622=1107.531,294.568,-77.936,-179.670,13.955,150.823
C00623=1107.525,294.320,-77.906,-179.675,13.954,150.823
C00624=1107.519,294.072,-77.876,-179.678,13.954,150.824
C00625=1107.514,293.824,-77.846,-179.682,13.953,150.825
C00626=1107.508,293.576,-77.816,-179.686,13.952,150.825
C00627=1107.502,293.327,-77.786,-179.690,13.951,150.826
C00628=1107.496,293.080,-77.756,-179.693,13.951,150.827
C00629=1107.491,292.831,-77.726,-179.698,13.950,150.828
C00630=1107.485,292.583,-77.696,-179.701,13.949,150.828
C00631=1107.479,292.335,-77.665,-179.705,13.949,150.829
C00632=1107.474,292.087,-77.636,-179.709,13.949,150.830
C00633=1107.468,291.839,-77.606,-179.713,13.948,150.830
C00634=1107.462,291.591,-77.576,-179.716,13.947,150.831
C00635=1107.457,291.342,-77.546,-179.720,13.947,150.832
C00636=1107.451,291.094,-77.516,-179.724,13.946,150.833
C00637=1107.446,290.846,-77.486,-179.728,13.945,150.833
C00638=1107.440,290.598,-77.456,-179.732,13.945,150.834
C00639=1107.435,290.350,-77.426,-179.735,13.945,150.835
C00640=1107.426,289.985,-77.383,-179.741,13.943,150.836
C00641=1107.418,289.621,-77.339,-179.747,13.943,150.837
C00642=1107.410,289.256,-77.295,-179.753,13.942,150.838
C00643=1107.401,288.891,-77.251,-179.758,13.941,150.839
C00644=1107.395,288.643,-77.221,-179.762,13.940,150.840
C00645=1107.389,288.395,-77.192,-179.766,13.940,150.841
C00646=1107.384,288.147,-77.162,-179.769,13.940,150.842
C00647=1107.378,287.899,-77.132,-179.773,13.939,150.842
C00648=1107.372,287.651,-77.102,-179.778,13.938,150.843
C00649=1107.367,287.403,-77.074,-179.781,13.938,150.844
C00650=1107.361,287.155,-77.044,-179.785,13.938,150.845
C00651=1107.355,286.907,-77.014,-179.789,13.937,150.845
C00652=1107.350,286.658,-76.984,-179.792,13.937,150.846
C00653=1107.343,286.410,-76.955,-179.797,13.936,150.847
C00654=1107.338,286.162,-76.925,-179.800,13.936,150.848
C00655=1107.332,285.913,-76.896,-179.804,13.935,150.848
C00656=1107.327,285.665,-76.866,-179.808,13.935,150.849
C00657=1107.321,285.418,-76.837,-179.812,13.934,150.850
C00658=1107.315,285.170,-76.807,-179.816,13.934,150.851
C00659=1107.310,284.921,-76.777,-179.820,13.933,150.851
C00660=1107.304,284.673,-76.748,-179.823,13.933,150.852
C00661=1107.298,284.425,-76.719,-179.827,13.933,150.853
C00662=1107.293,284.176,-76.689,-179.832,13.932,150.854
C00663=1107.287,283.929,-76.660,-179.835,13.931,150.855
C00664=1107.282,283.680,-76.631,-179.839,13.931,150.855
C00665=1107.276,283.432,-76.601,-179.843,13.931,150.856
C00666=1107.270,283.184,-76.572,-179.847,13.930,150.857
C00667=1107.264,282.935,-76.543,-179.851,13.930,150.858
C00668=1107.259,282.688,-76.513,-179.854,13.929,150.858
C00669=1107.253,282.440,-76.484,-179.858,13.929,150.859
C00670=1107.248,282.191,-76.455,-179.862,13.929,150.860
C00671=1107.242,281.943,-76.425,-179.866,13.928,150.861
C00672=1107.236,281.695,-76.396,-179.870,13.927,150.862
C00673=1107.231,281.447,-76.367,-179.874,13.927,150.862
C00674=1107.225,281.199,-76.338,-179.878,13.927,150.863
C00675=1107.219,280.950,-76.308,-179.881,13.926,150.864
C00676=1107.213,280.702,-76.279,-179.885,13.926,150.865
C00677=1107.208,280.454,-76.250,-179.890,13.926,150.866
C00678=1107.202,280.206,-76.221,-179.893,13.925,150.866
C00679=1107.197,279.957,-76.192,-179.897,13.925,150.867
C00680=1107.190,279.709,-76.163,-179.901,13.925,150.868
C00681=1107.185,279.461,-76.133,-179.904,13.924,150.869
C00682=1107.179,279.213,-76.104,-179.909,13.924,150.870
C00683=1107.174,278.965,-76.075,-179.913,13.923,150.870
C00684=1107.168,278.716,-76.046,-179.916,13.923,150.871
C00685=1107.162,278.468,-76.017,-179.920,13.923,150.872
C00686=1107.157,278.220,-75.988,-179.924,13.923,150.873
C00687=1107.151,277.972,-75.958,-179.928,13.923,150.874
C00688=1107.145,277.723,-75.930,-179.932,13.921,150.874
C00689=1107.139,277.475,-75.901,-179.936,13.921,150.875
C00690=1107.134,277.227,-75.872,-179.940,13.921,150.876
C00691=1107.128,276.978,-75.843,-179.944,13.921,150.877
C00692=1107.120,276.623,-75.801,-179.950,13.920,150.878
C00693=1107.112,276.269,-75.760,-179.955,13.920,150.879
C00694=1107.104,275.913,-75.719,-179.961,13.919,150.880
C00695=1107.096,275.558,-75.678,-179.966,13.919,150.882
C00696=1107.090,275.309,-75.648,-179.970,13.919,150.883
C00697=1107.085,275.061,-75.620,-179.974,13.919,150.883
C00698=1107.079,274.813,-75.591,-179.977,13.919,150.884
C00699=1107.073,274.564,-75.562,-179.982,13.918,150.885
C00700=1107.068,274.317,-75.534,-179.986,13.918,150.886
C00701=1107.061,274.069,-75.505,-179.990,13.918,150.887
C00702=1107.056,273.820,-75.476,-179.993,13.917,150.887
C00703=1107.051,273.572,-75.447,-179.997,13.917,150.888
C00704=1107.045,273.323,-75.419,179.999,13.917,150.889
C00705=1107.038,273.075,-75.390,179.995,13.917,150.890
C00706=1107.033,272.827,-75.362,179.990,13.916,150.891
C00707=1107.028,272.578,-75.333,179.987,13.916,150.892
C00708=1107.022,272.330,-75.304,179.983,13.916,150.893
C00709=1107.016,272.082,-75.276,179.979,13.915,150.893
C00710=1107.010,271.834,-75.247,179.975,13.915,150.894
C00711=1107.005,271.585,-75.218,179.971,13.915,150.895
C00712=1106.999,271.337,-75.189,179.968,13.915,150.896
C00713=1106.993,271.089,-75.161,179.964,13.915,150.897
C00714=1106.988,270.841,-75.133,179.959,13.914,150.898
C00715=1106.982,270.592,-75.104,179.955,13.914,150.898
C00716=1106.976,270.344,-75.076,179.951,13.914,150.899
C00717=1106.971,270.095,-75.047,179.947,13.914,150.900
C00718=1106.965,269.847,-75.018,179.944,13.914,150.901
C00719=1106.959,269.599,-74.990,179.940,13.914,150.902
C00720=1106.954,269.350,-74.962,179.936,13.913,150.903
C00721=1106.948,269.102,-74.934,179.932,13.913,150.903
C00722=1106.942,268.854,-74.905,179.928,13.913,150.904
C00723=1106.937,268.606,-74.877,179.925,13.913,150.905
C00724=1106.931,268.357,-74.848,179.920,13.912,150.906
C00725=1106.925,268.109,-74.820,179.916,13.912,150.907
C00726=1106.919,267.861,-74.791,179.912,13.912,150.908
C00727=1106.913,267.612,-74.763,179.908,13.912,150.909
C00728=1106.908,267.364,-74.735,179.904,13.912,150.909
C00729=1106.902,267.116,-74.707,179.901,13.912,150.910
C00730=1106.897,266.867,-74.678,179.897,13.912,150.911
C00731=1106.891,266.618,-74.650,179.893,13.912,150.912
C00732=1106.886,266.371,-74.621,179.889,13.912,150.913
C00733=1106.880,266.122,-74.593,179.885,13.912,150.914
C00734=1106.874,265.874,-74.565,179.881,13.912,150.915
C00735=1106.868,265.626,-74.537,179.877,13.912,150.916
C00736=1106.863,265.377,-74.509,179.873,13.911,150.916
C00737=1106.857,265.129,-74.480,179.869,13.911,150.917
C00738=1106.852,264.881,-74.452,179.865,13.911,150.918
C00739=1106.846,264.632,-74.424,179.861,13.911,150.919
C00740=1106.840,264.384,-74.397,179.857,13.911,150.920
C00741=1106.834,264.135,-74.368,179.853,13.911,150.921
C00742=1106.828,263.887,-74.341,179.849,13.911,150.922
C00743=1106.823,263.639,-74.312,179.845,13.911,150.923
C00744=1106.815,263.286,-74.272,179.840,13.911,150.924
C00745=1106.807,262.934,-74.233,179.834,13.910,150.925
C00746=1106.798,262.583,-74.193,179.828,13.911,150.927
C00747=1106.790,262.229,-74.154,179.823,13.911,150.928
C00748=1106.784,261.981,-74.126,179.819,13.911,150.929
C00749=1106.779,261.733,-74.098,179.815,13.911,150.930
C00750=1106.772,261.485,-74.070,179.811,13.911,150.931
C00751=1106.767,261.237,-74.042,179.807,13.911,150.931
C00752=1106.761,260.988,-74.014,179.802,13.910,150.932
C00753=1106.756,260.740,-73.986,179.799,13.910,150.933
C00754=1106.749,260.491,-73.959,179.794,13.910,150.934
C00755=1106.744,260.243,-73.931,179.791,13.910,150.935
C00756=1106.738,259.994,-73.903,179.787,13.910,150.936
C00757=1106.733,259.746,-73.875,179.783,13.910,150.937
C00758=1106.727,259.498,-73.847,179.779,13.910,150.938
C00759=1106.721,259.249,-73.820,179.775,13.910,150.939
C00760=1106.716,259.001,-73.792,179.771,13.910,150.940
C00761=1106.710,258.752,-73.763,179.767,13.910,150.940
C00762=1106.704,258.504,-73.736,179.763,13.910,150.941
C00763=1106.699,258.255,-73.709,179.759,13.910,150.942
C00764=1106.693,258.007,-73.680,179.755,13.910,150.943
C00765=1106.687,257.759,-73.653,179.751,13.910,150.944
C00766=1106.681,257.510,-73.625,179.747,13.910,150.945
C00767=1106.676,257.262,-73.597,179.743,13.910,150.946
C00768=1106.669,257.014,-73.570,179.739,13.910,150.947
C00769=1106.664,256.764,-73.543,179.735,13.911,150.948
C00770=1106.659,256.516,-73.515,179.731,13.911,150.949
C00771=1106.653,256.268,-73.488,179.727,13.910,150.950
C00772=1106.647,256.019,-73.460,179.723,13.910,150.950
C00773=1106.641,255.772,-73.432,179.720,13.910,150.951
C00774=1106.636,255.523,-73.405,179.715,13.911,150.952
C00775=1106.630,255.274,-73.377,179.711,13.911,150.953
C00776=1106.624,255.026,-73.350,179.708,13.911,150.954
C00777=1106.619,254.778,-73.322,179.704,13.911,150.955
C00778=1106.613,254.529,-73.295,179.699,13.911,150.956
C00779=1106.607,254.281,-73.267,179.696,13.911,150.957
C00780=1106.602,254.032,-73.240,179.692,13.911,150.958
C00781=1106.596,253.784,-73.212,179.688,13.911,150.959
C00782=1106.590,253.535,-73.185,179.684,13.911,150.960
C00783=1106.584,253.287,-73.158,179.680,13.911,150.961
C00784=1106.579,253.038,-73.130,179.676,13.911,150.961
C00785=1106.573,252.790,-73.104,179.672,13.911,150.962
C00786=1106.567,252.541,-73.075,179.668,13.911,150.963
C00787=1106.562,252.293,-73.049,179.664,13.911,150.964
C00788=1106.556,252.045,-73.021,179.660,13.911,150.965
C00789=1106.550,251.797,-72.994,179.656,13.911,150.966
C00790=1106.545,251.548,-72.967,179.652,13.912,150.967
C00791=1106.539,251.299,-72.939,179.648,13.912,150.968
C00792=1106.534,251.051,-72.912,179.644,13.912,150.969
C00793=1106.528,250.802,-72.885,179.640,13.912,150.970
C00794=1106.523,250.554,-72.858,179.636,13.912,150.971
C00795=1106.516,250.305,-72.830,179.632,13.912,150.972
C00796=1106.509,249.950,-72.792,179.626,13.912,150.973
C00797=1106.501,249.595,-72.752,179.620,13.912,150.974
C00798=1106.493,249.240,-72.714,179.615,13.912,150.976
C00799=1106.485,248.885,-72.676,179.609,13.912,150.977
C00800=1106.479,248.637,-72.648,179.605,13.913,150.978
C00801=1106.473,248.388,-72.621,179.601,13.913,150.979
C00802=1106.468,248.139,-72.594,179.597,13.913,150.980
C00803=1106.462,247.891,-72.567,179.594,13.913,150.981
C00804=1106.457,247.643,-72.540,179.589,13.913,150.982
C00805=1106.452,247.394,-72.513,179.585,13.913,150.983
C00806=1106.445,247.146,-72.486,179.582,13.913,150.983
C00807=1106.439,246.897,-72.459,179.577,13.913,150.984
C00808=1106.434,246.649,-72.432,179.573,13.913,150.985
C00809=1106.428,246.400,-72.405,179.569,13.914,150.986
C00810=1106.423,246.152,-72.378,179.565,13.914,150.987
C00811=1106.417,245.903,-72.351,179.561,13.914,150.988
C00812=1106.412,245.655,-72.324,179.557,13.914,150.989
C00813=1106.406,245.407,-72.298,179.553,13.914,150.990
C00814=1106.400,245.158,-72.271,179.549,13.914,150.991
C00815=1106.395,244.909,-72.243,179.546,13.915,150.992
C00816=1106.389,244.660,-72.217,179.542,13.915,150.993
C00817=1106.383,244.412,-72.190,179.538,13.915,150.994
C00818=1106.377,244.164,-72.163,179.534,13.915,150.995
C00819=1106.372,243.915,-72.136,179.530,13.915,150.996
C00820=1106.366,243.667,-72.110,179.526,13.916,150.997
C00821=1106.361,243.418,-72.083,179.522,13.916,150.998
C00822=1106.355,243.170,-72.056,179.518,13.916,150.999
C00823=1106.349,242.922,-72.030,179.514,13.916,151.000
C00824=1106.344,242.673,-72.002,179.510,13.916,151.001
C00825=1106.339,242.424,-71.976,179.506,13.916,151.002
C00826=1106.333,242.176,-71.950,179.501,13.917,151.003
C00827=1106.326,241.927,-71.923,179.498,13.917,151.003
C00828=1106.321,241.678,-71.896,179.494,13.917,151.004
C00829=1106.315,241.430,-71.870,179.489,13.917,151.005
C00830=1106.309,241.181,-71.843,179.485,13.917,151.006
C00831=1106.304,240.932,-71.817,179.482,13.918,151.007
C00832=1106.298,240.684,-71.790,179.478,13.918,151.008
C00833=1106.292,240.436,-71.764,179.474,13.919,151.009
C00834=1106.286,240.187,-71.737,179.470,13.919,151.010
C00835=1106.281,239.939,-71.710,179.466,13.919,151.011
C00836=1106.275,239.690,-71.684,179.462,13.919,151.012
C00837=1106.269,239.442,-71.658,179.458,13.919,151.013
C00838=1106.264,239.193,-71.631,179.454,13.919,151.014
C00839=1106.258,238.944,-71.605,179.449,13.920,151.015
C00840=1106.252,238.696,-71.579,179.446,13.920,151.016
C00841=1106.247,238.448,-71.552,179.441,13.920,151.017
C00842=1106.241,238.199,-71.526,179.438,13.921,151.018
C00843=1106.235,237.950,-71.499,179.434,13.921,151.019
C00844=1106.229,237.702,-71.473,179.430,13.921,151.020
C00845=1106.224,237.453,-71.447,179.426,13.922,151.021
C00846=1106.218,237.205,-71.420,179.422,13.922,151.022
C00847=1106.212,236.956,-71.393,179.418,13.922,151.023
C00848=1106.205,236.595,-71.355,179.412,13.923,151.024
C00849=1106.196,236.233,-71.317,179.406,13.923,151.026
C00850=1106.188,235.871,-71.279,179.400,13.923,151.027
C00851=1106.180,235.509,-71.240,179.394,13.923,151.029
C00852=1106.174,235.260,-71.214,179.390,13.923,151.029
C00853=1106.169,235.012,-71.188,179.386,13.924,151.030
C00854=1106.163,234.764,-71.162,179.383,13.925,151.032
C00855=1106.157,234.515,-71.136,179.379,13.925,151.032
C00856=1106.152,234.266,-71.110,179.375,13.925,151.033
C00857=1106.146,234.018,-71.084,179.371,13.925,151.034
C00858=1106.140,233.769,-71.057,179.366,13.926,151.035
C00859=1106.135,233.520,-71.031,179.363,13.926,151.036
C00860=1106.129,233.271,-71.005,179.358,13.926,151.037
C00861=1106.123,233.023,-70.979,179.354,13.926,151.038
C00862=1106.117,232.774,-70.953,179.351,13.927,151.039
C00863=1106.112,232.527,-70.927,179.347,13.927,151.040
C00864=1106.107,232.278,-70.901,179.343,13.928,151.041
C00865=1106.101,232.029,-70.876,179.339,13.928,151.042
C00866=1106.095,231.780,-70.849,179.335,13.928,151.043
C00867=1106.089,231.532,-70.823,179.330,13.929,151.044
C00868=1106.084,231.283,-70.797,179.327,13.929,151.045
C00869=1106.078,231.034,-70.770,179.322,13.929,151.046
C00870=1106.072,230.786,-70.746,179.319,13.930,151.047
C00871=1106.067,230.537,-70.720,179.315,13.930,151.048
C00872=1106.061,230.289,-70.693,179.311,13.931,151.049
C00873=1106.055,230.040,-70.668,179.307,13.931,151.050
C00874=1106.050,229.791,-70.642,179.303,13.931,151.051
C00875=1106.044,229.542,-70.616,179.299,13.931,151.052
C00876=1106.038,229.294,-70.590,179.294,13.931,151.053
C00877=1106.033,229.046,-70.564,179.291,13.933,151.054
C00878=1106.027,228.797,-70.538,179.287,13.933,151.055
C00879=1106.021,228.548,-70.513,179.283,13.933,151.056
C00880=1106.016,228.299,-70.487,179.279,13.933,151.057
C00881=1106.009,228.051,-70.462,179.275,13.933,151.058
C00882=1106.004,227.802,-70.435,179.270,13.934,151.059
C00883=1105.999,227.554,-70.409,179.267,13.935,151.060
C00884=1105.992,227.305,-70.384,179.263,13.935,151.061
C00885=1105.987,227.056,-70.358,179.259,13.935,151.062
C00886=1105.981,226.808,-70.333,179.255,13.935,151.063
C00887=1105.975,226.559,-70.307,179.251,13.936,151.064
C00888=1105.970,226.311,-70.282,179.246,13.936,151.065
C00889=1105.964,226.062,-70.256,179.243,13.937,151.066
C00890=1105.959,225.813,-70.230,179.239,13.937,151.067
C00891=1105.953,225.564,-70.205,179.235,13.938,151.068
C00892=1105.948,225.316,-70.179,179.231,13.938,151.069
C00893=1105.942,225.067,-70.154,179.227,13.938,151.070
C00894=1105.936,224.818,-70.128,179.223,13.938,151.071
C00895=1105.930,224.569,-70.102,179.219,13.939,151.072
C00896=1105.925,224.321,-70.077,179.215,13.940,151.073
C00897=1105.919,224.073,-70.052,179.211,13.940,151.074
C00898=1105.913,223.824,-70.026,179.207,13.940,151.075
C00899=1105.908,223.576,-70.001,179.203,13.941,151.076
C00900=1105.899,223.205,-69.962,179.197,13.941,151.078
C00901=1105.890,222.835,-69.925,179.191,13.942,151.079
C00902=1105.883,222.466,-69.886,179.185,13.943,151.081
C00903=1105.874,222.095,-69.849,179.180,13.944,151.082
C00904=1105.868,221.847,-69.824,179.175,13.944,151.083
C00905=1105.862,221.598,-69.798,179.171,13.945,151.084
C00906=1105.857,221.349,-69.772,179.167,13.945,151.085
C00907=1105.851,221.101,-69.748,179.163,13.945,151.086
C00908=1105.845,220.852,-69.723,179.159,13.946,151.087
C00909=1105.840,220.603,-69.697,179.156,13.946,151.088
C00910=1105.834,220.355,-69.672,179.151,13.947,151.089
C00911=1105.828,220.106,-69.647,179.147,13.947,151.090
C00912=1105.823,219.857,-69.621,179.143,13.947,151.091
C00913=1105.817,219.609,-69.596,179.140,13.948,151.092
C00914=1105.811,219.360,-69.571,179.135,13.949,151.093
C00915=1105.805,219.111,-69.545,179.131,13.949,151.094
C00916=1105.800,218.862,-69.521,179.127,13.949,151.095
C00917=1105.794,218.614,-69.495,179.123,13.950,151.096
C00918=1105.788,218.365,-69.470,179.120,13.951,151.097
C00919=1105.783,218.116,-69.445,179.116,13.951,151.098
C00920=1105.777,217.868,-69.420,179.111,13.951,151.099
C00921=1105.771,217.620,-69.395,179.107,13.952,151.100
C00922=1105.765,217.370,-69.370,179.103,13.952,151.101
C00923=1105.760,217.121,-69.344,179.100,13.953,151.102
C00924=1105.755,216.873,-69.320,179.095,13.953,151.103
C00925=1105.748,216.624,-69.295,179.091,13.954,151.104
C00926=1105.743,216.376,-69.270,179.087,13.954,151.105
C00927=1105.738,216.127,-69.245,179.084,13.955,151.106
C00928=1105.732,215.879,-69.220,179.080,13.955,151.107
C00929=1105.726,215.629,-69.195,179.076,13.956,151.108
C00930=1105.720,215.381,-69.170,179.071,13.956,151.109
C00931=1105.715,215.132,-69.145,179.067,13.956,151.111
C00932=1105.709,214.883,-69.120,179.064,13.958,151.112
C00933=1105.704,214.634,-69.095,179.060,13.958,151.112
C00934=1105.698,214.386,-69.070,179.056,13.958,151.114
C00935=1105.692,214.137,-69.046,179.051,13.959,151.115
C00936=1105.686,213.889,-69.020,179.048,13.959,151.116
C00937=1105.681,213.640,-68.996,179.044,13.960,151.117
C00938=1105.675,213.391,-68.970,179.040,13.960,151.118
C00939=1105.670,213.142,-68.946,179.036,13.960,151.119
C00940=1105.664,212.894,-68.921,179.032,13.961,151.120
C00941=1105.659,212.645,-68.896,179.028,13.962,151.121
C00942=1105.653,212.396,-68.872,179.024,13.962,151.122
C00943=1105.647,212.148,-68.847,179.020,13.962,151.123
C00944=1105.641,211.899,-68.822,179.016,13.963,151.124
C00945=1105.636,211.651,-68.797,179.012,13.964,151.125
C00946=1105.630,211.401,-68.772,179.008,13.965,151.126
C00947=1105.624,211.153,-68.748,179.004,13.965,151.127
C00948=1105.618,210.904,-68.723,179.000,13.965,151.128
C00949=1105.613,210.655,-68.699,178.996,13.966,151.129
C00950=1105.607,210.406,-68.674,178.992,13.967,151.130
C00951=1105.602,210.158,-68.650,178.988,13.967,151.131
C00952=1105.593,209.791,-68.613,178.982,13.968,151.132
C00953=1105.584,209.424,-68.577,178.976,13.968,151.134
C00954=1105.577,209.058,-68.540,178.970,13.970,151.135
C00955=1105.568,208.691,-68.504,178.965,13.970,151.137
C00956=1105.545,207.696,-68.407,178.940,13.971,151.143
C00957=1105.539,207.447,-68.382,178.936,13.973,151.144
C00958=1105.534,207.198,-68.358,178.931,13.974,151.145
C00959=1105.528,206.949,-68.333,178.927,13.976,151.147
C00960=1105.522,206.701,-68.309,178.922,13.977,151.148
C00961=1105.516,206.451,-68.285,178.918,13.978,151.149
C00962=1105.511,206.203,-68.260,178.914,13.979,151.150
C00963=1105.505,205.954,-68.236,178.910,13.981,151.152
C00964=1105.499,205.705,-68.212,178.906,13.982,151.153
C00965=1105.493,205.457,-68.188,178.901,13.984,151.154
C00966=1105.488,205.208,-68.164,178.897,13.985,151.156
C00967=1105.482,204.959,-68.139,178.893,13.986,151.157
C00968=1105.477,204.710,-68.115,178.889,13.988,151.158
C00969=1105.471,204.462,-68.091,178.884,13.989,151.159
C00970=1105.465,204.213,-68.066,178.881,13.990,151.161
C00971=1105.460,203.964,-68.042,178.876,13.991,151.162
C00972=1105.454,203.716,-68.018,178.872,13.993,151.163
C00973=1105.448,203.467,-67.994,178.868,13.994,151.164
C00974=1105.442,203.218,-67.970,178.864,13.995,151.166
C00975=1105.437,202.969,-67.945,178.859,13.996,151.167
C00976=1105.431,202.720,-67.921,178.855,13.998,151.168
C00977=1105.425,202.472,-67.897,178.850,13.999,151.169
C00978=1105.419,202.223,-67.873,178.846,14.001,151.171
C00979=1105.413,201.974,-67.849,178.842,14.002,151.172
C00980=1105.408,201.726,-67.825,178.838,14.003,151.173
C00981=1105.402,201.476,-67.801,178.833,14.004,151.174
C00982=1105.396,201.227,-67.777,178.830,14.006,151.176
C00983=1105.390,200.979,-67.753,178.826,14.007,151.177
C00984=1105.384,200.730,-67.729,178.821,14.008,151.178
C00985=1105.378,200.482,-67.705,178.817,14.010,151.179
C00986=1105.373,200.233,-67.681,178.813,14.011,151.181
C00987=1105.367,199.983,-67.658,178.808,14.013,151.182
C00988=1105.361,199.735,-67.633,178.804,14.014,151.183
C00989=1105.355,199.487,-67.610,178.800,14.015,151.185
C00990=1105.350,199.238,-67.585,178.795,14.016,151.186
C00991=1105.345,198.988,-67.561,178.792,14.018,151.187
C00992=1105.339,198.740,-67.538,178.787,14.019,151.188
C00993=1105.332,198.492,-67.514,178.783,14.021,151.189
C00994=1105.327,198.243,-67.490,178.779,14.021,151.191
C00995=1105.321,197.993,-67.467,178.775,14.023,151.192
C00996=1105.316,197.745,-67.442,178.770,14.024,151.193
C00997=1105.310,197.496,-67.419,178.766,14.026,151.194
C00998=1105.305,197.247,-67.395,178.762,14.027,151.196
C00999=1105.298,196.998,-67.371,178.758,14.028,151.197
C01000=1105.293,196.750,-67.347,178.754,14.029,151.198
C01001=1105.287,196.501,-67.324,178.750,14.030,151.199
C01002=1105.282,196.252,-67.300,178.746,14.032,151.201
C01003=1105.275,196.003,-67.276,178.741,14.033,151.202
C01004=1105.270,195.754,-67.252,178.737,14.035,151.203
C01005=1105.264,195.506,-67.228,178.733,14.035,151.204
C01006=1105.258,195.257,-67.205,178.729,14.037,151.205
C01007=1105.253,195.008,-67.181,178.724,14.038,151.207
C01008=1105.247,194.759,-67.158,178.721,14.040,151.208
C01009=1105.241,194.510,-67.134,178.716,14.040,151.209
C01010=1105.236,194.261,-67.111,178.713,14.042,151.210
C01011=1105.229,194.013,-67.087,178.708,14.043,151.212
C01012=1105.224,193.764,-67.063,178.704,14.044,151.213
C01013=1105.218,193.515,-67.040,178.699,14.045,151.214
C01014=1105.213,193.266,-67.016,178.696,14.047,151.215
C01015=1105.207,193.017,-66.992,178.692,14.048,151.216
C01016=1105.201,192.768,-66.969,178.688,14.049,151.218
C01017=1105.195,192.497,-66.944,178.683,14.051,151.219
C01018=1105.189,192.226,-66.918,178.679,14.052,151.220
C01019=1105.183,191.956,-66.892,178.674,14.053,151.222
C01020=1105.176,191.684,-66.867,178.669,14.055,151.223
C01021=1105.171,191.436,-66.844,178.665,14.056,151.224
C01022=1105.165,191.187,-66.819,178.661,14.057,151.225
C01023=1105.160,190.938,-66.796,178.657,14.058,151.226
C01024=1105.154,190.689,-66.773,178.653,14.059,151.228
C01025=1105.148,190.441,-66.749,178.649,14.061,151.229
C01026=1105.143,190.192,-66.726,178.645,14.062,151.230
C01027=1105.137,189.943,-66.703,178.641,14.063,151.231
C01028=1105.131,189.695,-66.680,178.637,14.065,151.233
C01029=1105.126,189.445,-66.656,178.633,14.065,151.234
C01030=1105.120,189.196,-66.633,178.629,14.067,151.235
C01031=1105.115,188.948,-66.610,178.624,14.068,151.236
C01032=1105.109,188.699,-66.586,178.621,14.069,151.237
C01033=1105.103,188.449,-66.563,178.616,14.070,151.238
C01034=1105.097,188.200,-66.540,178.612,14.072,151.240
C01035=1105.091,187.952,-66.517,178.608,14.072,151.241
C01036=1105.086,187.702,-66.493,178.604,14.074,151.242
C01037=1105.080,187.454,-66.470,178.600,14.075,151.243
C01038=1105.075,187.205,-66.447,178.596,14.076,151.244
C01039=1105.069,186.956,-66.424,178.592,14.077,151.246
C01040=1105.063,186.707,-66.401,178.588,14.078,151.247
C01041=1105.058,186.458,-66.377,178.583,14.079,151.248
C01042=1105.052,186.209,-66.354,178.580,14.081,151.249
C01043=1105.047,185.962,-66.331,178.575,14.082,151.250
C01044=1105.041,185.713,-66.308,178.572,14.083,151.251
C01045=1105.036,185.464,-66.285,178.567,14.084,151.253
C01046=1105.031,185.215,-66.262,178.564,14.085,151.254
C01047=1105.025,184.966,-66.239,178.560,14.087,151.255
C01048=1105.019,184.717,-66.216,178.555,14.088,151.256
C01049=1105.013,184.467,-66.192,178.552,14.089,151.257
C01050=1105.007,184.218,-66.169,178.547,14.090,151.258
C01051=1105.001,183.970,-66.147,178.543,14.092,151.260
C01052=1104.995,183.721,-66.124,178.539,14.092,151.261
C01053=1104.989,183.472,-66.101,178.535,14.094,151.262
C01054=1104.983,183.223,-66.078,178.531,14.095,151.263
C01055=1104.978,182.974,-66.055,178.527,14.096,151.264
C01056=1104.972,182.725,-66.032,178.523,14.097,151.266
C01057=1104.966,182.476,-66.009,178.519,14.098,151.267
C01058=1104.960,182.228,-65.986,178.515,14.100,151.268
C01059=1104.955,181.979,-65.963,178.511,14.101,151.269
C01060=1104.949,181.730,-65.940,178.507,14.102,151.270
C01061=1104.943,181.481,-65.918,178.503,14.103,151.271
C01062=1104.938,181.232,-65.895,178.499,14.104,151.273
C01063=1104.931,180.983,-65.872,178.494,14.105,151.274
C01064=1104.925,180.734,-65.849,178.491,14.107,151.275
C01065=1104.920,180.486,-65.826,178.486,14.108,151.276
C01066=1104.914,180.237,-65.803,178.483,14.109,151.277
C01067=1104.909,179.988,-65.781,178.478,14.110,151.278
C01068=1104.903,179.739,-65.759,178.475,14.111,151.279
C01069=1104.898,179.490,-65.736,178.471,14.113,151.281
C01070=1104.891,179.241,-65.713,178.467,14.113,151.282
C01071=1104.885,178.993,-65.690,178.463,14.115,151.283
C01072=1104.880,178.744,-65.667,178.459,14.116,151.284
C01073=1104.874,178.495,-65.644,178.455,14.117,151.285
C01074=1104.869,178.245,-65.622,178.450,14.118,151.286
C01075=1104.863,177.996,-65.599,178.447,14.119,151.288
C01076=1104.856,177.748,-65.577,178.442,14.120,151.289
C01077=1104.851,177.499,-65.554,178.439,14.121,151.290
C01078=1104.846,177.250,-65.532,178.434,14.122,151.291
C01079=1104.840,177.001,-65.509,178.431,14.124,151.292
C01080=1104.834,176.752,-65.486,178.426,14.124,151.293
C01081=1104.828,176.481,-65.462,178.423,14.126,151.295
C01082=1104.822,176.209,-65.438,178.418,14.127,151.296
C01083=1104.816,175.938,-65.413,178.413,14.128,151.297
C01084=1104.809,175.667,-65.388,178.410,14.130,151.298
C01085=1104.803,175.417,-65.366,178.405,14.130,151.299
C01086=1104.798,175.169,-65.343,178.402,14.132,151.301
C01087=1104.792,174.920,-65.320,178.397,14.132,151.302
C01088=1104.786,174.671,-65.299,178.394,14.134,151.303
C01089=1104.780,174.422,-65.276,178.389,14.135,151.304
C01090=1104.775,174.173,-65.254,178.386,14.136,151.305
C01091=1104.770,173.924,-65.231,178.382,14.137,151.306
C01092=1104.763,173.676,-65.209,178.378,14.138,151.307
C01093=1104.758,173.426,-65.186,178.374,14.139,151.308
C01094=1104.752,173.177,-65.163,178.370,14.140,151.310
C01095=1104.746,172.928,-65.142,178.366,14.141,151.311
C01096=1104.741,172.680,-65.119,178.362,14.142,151.312
C01097=1104.735,172.430,-65.097,178.358,14.144,151.313
C01098=1104.729,172.182,-65.075,178.354,14.144,151.314
C01099=1104.724,171.932,-65.052,178.350,14.145,151.315
C01100=1104.718,171.684,-65.030,178.346,14.146,151.316
C01101=1104.712,171.435,-65.008,178.343,14.147,151.317
C01102=1104.707,171.186,-64.985,178.338,14.148,151.319
C01103=1104.701,170.937,-64.963,178.335,14.150,151.320
C01104=1104.695,170.689,-64.941,178.331,14.151,151.321
C01105=1104.690,170.439,-64.919,178.327,14.151,151.322
C01106=1104.684,170.190,-64.897,178.323,14.153,151.323
C01107=1104.678,169.941,-64.874,178.319,14.153,151.324
C01108=1104.673,169.692,-64.852,178.316,14.155,151.325
C01109=1104.667,169.444,-64.830,178.311,14.155,151.326
C01110=1104.661,169.194,-64.808,178.307,14.157,151.327
C01111=1104.656,168.945,-64.786,178.303,14.158,151.328
C01112=1104.650,168.697,-64.764,178.300,14.159,151.329
C01113=1104.644,168.447,-64.741,178.295,14.159,151.331
C01114=1104.639,168.199,-64.720,178.292,14.161,151.332
C01115=1104.633,167.950,-64.697,178.288,14.161,151.333
C01116=1104.628,167.700,-64.675,178.284,14.163,151.334
C01117=1104.622,167.452,-64.654,178.281,14.164,151.335
C01118=1104.617,167.202,-64.631,178.276,14.164,151.336
C01119=1104.610,166.954,-64.609,178.273,14.166,151.337
C01120=1104.605,166.705,-64.587,178.269,14.166,151.338
C01121=1104.599,166.456,-64.566,178.265,14.168,151.339
C01122=1104.594,166.206,-64.543,178.261,14.168,151.340
C01123=1104.588,165.958,-64.521,178.257,14.170,151.341
C01124=1104.583,165.709,-64.499,178.253,14.170,151.342
C01125=1104.577,165.460,-64.478,178.250,14.171,151.344
C01126=1104.572,165.211,-64.456,178.245,14.172,151.345
C01127=1104.565,164.962,-64.434,178.242,14.173,151.346
C01128=1104.560,164.713,-64.411,178.238,14.174,151.347
C01129=1104.554,164.464,-64.390,178.234,14.175,151.348
C01130=1104.549,164.215,-64.368,178.231,14.176,151.349
C01131=1104.543,163.966,-64.346,178.227,14.177,151.350
C01132=1104.538,163.717,-64.324,178.223,14.178,151.351
C01133=1104.532,163.468,-64.303,178.219,14.179,151.352
C01134=1104.527,163.219,-64.281,178.215,14.180,151.353
C01135=1104.521,162.970,-64.259,178.211,14.180,151.354
C01136=1104.515,162.721,-64.236,178.208,14.181,151.355
C01137=1104.510,162.473,-64.215,178.204,14.182,151.356
C01138=1104.504,162.223,-64.193,178.200,14.183,151.357
C01139=1104.499,161.975,-64.172,178.196,14.184,151.358
C01140=1104.493,161.725,-64.149,178.193,14.185,151.359
C01141=1104.488,161.477,-64.128,178.188,14.186,151.360
C01142=1104.482,161.227,-64.106,178.185,14.187,151.361
C01143=1104.476,160.978,-64.084,178.182,14.188,151.362
C01144=1104.471,160.729,-64.063,178.177,14.189,151.364
C01145=1104.464,160.457,-64.040,178.173,14.190,151.365
C01146=1104.458,160.185,-64.016,178.169,14.191,151.366
C01147=1104.452,159.914,-63.992,178.165,14.192,151.367
C01148=1104.446,159.642,-63.969,178.160,14.193,151.368
C01149=1104.440,159.393,-63.947,178.157,14.194,151.369
C01150=1104.434,159.144,-63.925,178.154,14.195,151.370
C01151=1104.428,158.896,-63.904,178.149,14.195,151.371
C01152=1104.423,158.646,-63.882,178.146,14.197,151.372
C01153=1104.418,158.397,-63.861,178.142,14.197,151.373
C01154=1104.411,158.148,-63.840,178.138,14.199,151.375
C01155=1104.406,157.899,-63.818,178.134,14.199,151.375
C01156=1104.400,157.650,-63.796,178.131,14.200,151.377
C01157=1104.395,157.401,-63.775,178.127,14.201,151.378
C01158=1104.389,157.152,-63.753,178.123,14.202,151.379
C01159=1104.383,156.903,-63.732,178.119,14.202,151.380
C01160=1104.377,156.654,-63.711,178.116,14.204,151.381
C01161=1104.372,156.405,-63.690,178.112,14.205,151.382
C01162=1104.366,156.156,-63.668,178.108,14.205,151.383
C01163=1104.361,155.907,-63.646,178.105,14.206,151.384
C01164=1104.355,155.658,-63.625,178.100,14.207,151.385
C01165=1104.349,155.409,-63.604,178.097,14.208,151.386
C01166=1104.343,155.160,-63.583,178.093,14.209,151.387
C01167=1104.338,154.911,-63.561,178.089,14.210,151.388
C01168=1104.331,154.662,-63.540,178.086,14.210,151.389
C01169=1104.326,154.413,-63.519,178.082,14.211,151.390
C01170=1104.321,154.164,-63.498,178.079,14.213,151.391
C01171=1104.315,153.915,-63.476,178.075,14.213,151.392
C01172=1104.310,153.666,-63.455,178.071,14.214,151.393
C01173=1104.304,153.416,-63.433,178.067,14.215,151.394
C01174=1104.298,153.168,-63.412,178.064,14.216,151.395
C01175=1104.292,152.918,-63.391,178.059,14.216,151.396
C01176=1104.287,152.670,-63.370,178.056,14.217,151.397
C01177=1104.281,152.421,-63.349,178.052,14.218,151.398
C01178=1104.275,152.171,-63.328,178.049,14.219,151.399
C01179=1104.270,151.923,-63.306,178.045,14.220,151.400
C01180=1104.264,151.674,-63.285,178.041,14.221,151.401
C01181=1104.258,151.424,-63.264,178.038,14.222,151.402
C01182=1104.252,151.175,-63.243,178.034,14.222,151.403
C01183=1104.247,150.926,-63.222,178.031,14.223,151.404
C01184=1104.241,150.678,-63.201,178.026,14.224,151.405
C01185=1104.235,150.428,-63.180,178.023,14.225,151.406
C01186=1104.230,150.179,-63.159,178.019,14.225,151.407
C01187=1104.225,149.930,-63.138,178.016,14.226,151.408
C01188=1104.219,149.681,-63.116,178.011,14.227,151.409
C01189=1104.213,149.432,-63.096,178.008,14.228,151.410
C01190=1104.207,149.183,-63.074,178.005,14.229,151.411
C01191=1104.202,148.933,-63.054,178.001,14.229,151.412
C01192=1104.196,148.685,-63.032,177.997,14.231,151.413
C01193=1104.190,148.435,-63.012,177.993,14.231,151.414
C01194=1104.184,148.187,-62.991,177.990,14.232,151.415
C01195=1104.179,147.938,-62.970,177.986,14.232,151.416
C01196=1104.173,147.689,-62.949,177.982,14.234,151.417
C01197=1104.167,147.439,-62.928,177.979,14.235,151.418
C01198=1104.162,147.191,-62.907,177.975,14.235,151.419
C01199=1104.156,146.941,-62.886,177.972,14.236,151.420
C01200=1104.150,146.692,-62.866,177.968,14.236,151.421
C01201=1104.144,146.444,-62.845,177.964,14.238,151.422
C01202=1104.139,146.194,-62.824,177.961,14.238,151.423
C01203=1104.133,145.946,-62.802,177.957,14.239,151.424
C01204=1104.128,145.696,-62.782,177.953,14.239,151.425
C01205=1104.121,145.447,-62.762,177.950,14.240,151.426
C01206=1104.116,145.198,-62.740,177.946,14.242,151.427
C01207=1104.110,144.949,-62.720,177.942,14.242,151.428
C01208=1104.105,144.699,-62.699,177.939,14.243,151.429
C01209=1104.099,144.428,-62.676,177.935,14.243,151.430
C01210=1104.092,144.156,-62.654,177.931,14.244,151.431
C01211=1104.086,143.883,-62.631,177.927,14.245,151.432
C01212=1104.080,143.612,-62.608,177.923,14.246,151.433
C01213=1104.075,143.363,-62.588,177.920,14.247,151.434
C01214=1104.068,143.113,-62.567,177.916,14.247,151.435
C01215=1104.063,142.864,-62.547,177.913,14.248,151.436
C01216=1104.057,142.616,-62.526,177.909,14.249,151.437
C01217=1104.052,142.367,-62.505,177.905,14.250,151.438
C01218=1104.045,142.117,-62.485,177.901,14.250,151.439
C01219=1104.040,141.868,-62.464,177.898,14.251,151.440
C01220=1104.035,141.619,-62.444,177.894,14.252,151.441
C01221=1104.029,141.370,-62.422,177.891,14.252,151.442
C01222=1104.023,141.121,-62.402,177.888,14.253,151.443
C01223=1104.017,140.872,-62.381,177.884,14.254,151.444
C01224=1104.012,140.623,-62.361,177.881,14.254,151.444
C01225=1104.006,140.374,-62.341,177.876,14.255,151.446
C01226=1104.001,140.125,-62.320,177.873,14.256,151.446
C01227=1103.995,139.875,-62.299,177.869,14.256,151.447
C01228=1103.989,139.626,-62.280,177.866,14.257,151.448
C01229=1103.983,139.377,-62.258,177.863,14.258,151.449
C01230=1103.977,139.129,-62.238,177.859,14.258,151.450
C01231=1103.972,138.879,-62.218,177.855,14.260,151.451
C01232=1103.966,138.630,-62.197,177.852,14.260,151.452
C01233=1103.960,138.381,-62.177,177.848,14.261,151.453
C01234=1103.955,138.132,-62.156,177.844,14.261,151.454
C01235=1103.949,137.883,-62.136,177.841,14.262,151.455
C01236=1103.944,137.634,-62.116,177.837,14.262,151.456
C01237=1103.937,137.384,-62.095,177.834,14.263,151.457
C01238=1103.932,137.135,-62.075,177.831,14.264,151.458
C01239=1103.926,136.886,-62.055,177.827,14.265,151.459
C01240=1103.921,136.637,-62.034,177.824,14.266,151.460
C01241=1103.915,136.388,-62.014,177.820,14.266,151.461
C01242=1103.910,136.139,-61.994,177.816,14.267,151.461
C01243=1103.904,135.890,-61.974,177.813,14.267,151.462
C01244=1103.898,135.641,-61.953,177.809,14.268,151.463
C01245=1103.892,135.391,-61.934,177.806,14.269,151.464
C01246=1103.887,135.142,-61.913,177.802,14.269,151.465
C01247=1103.881,134.893,-61.893,177.799,14.270,151.466
C01248=1103.875,134.644,-61.873,177.795,14.270,151.467
C01249=1103.870,134.395,-61.853,177.792,14.271,151.468
C01250=1103.864,134.146,-61.832,177.788,14.271,151.469
C01251=1103.858,133.897,-61.812,177.785,14.272,151.470
C01252=1103.852,133.648,-61.791,177.782,14.273,151.471
C01253=1103.847,133.398,-61.772,177.778,14.274,151.472
C01254=1103.841,133.149,-61.752,177.775,14.274,151.472
C01255=1103.835,132.900,-61.732,177.771,14.275,151.473
C01256=1103.830,132.651,-61.711,177.768,14.276,151.474
C01257=1103.824,132.402,-61.691,177.764,14.275,151.475
C01258=1103.819,132.153,-61.672,177.761,14.276,151.476
C01259=1103.813,131.904,-61.651,177.758,14.277,151.477
C01260=1103.807,131.655,-61.631,177.754,14.277,151.478
C01261=1103.801,131.406,-61.611,177.751,14.278,151.479
C01262=1103.796,131.156,-61.591,177.747,14.279,151.480
C01263=1103.790,130.907,-61.571,177.743,14.280,151.481
C01264=1103.784,130.658,-61.551,177.740,14.280,151.482
C01265=1103.778,130.409,-61.531,177.736,14.281,151.482
C01266=1103.773,130.159,-61.511,177.733,14.282,151.483
C01267=1103.767,129.911,-61.491,177.729,14.282,151.484
C01268=1103.761,129.662,-61.471,177.726,14.283,151.485
C01269=1103.756,129.412,-61.452,177.722,14.283,151.486
C01270=1103.750,129.163,-61.432,177.719,14.284,151.487
C01271=1103.744,128.914,-61.412,177.715,14.284,151.488
C01272=1103.738,128.665,-61.392,177.712,14.285,151.489
C01273=1103.731,128.393,-61.370,177.708,14.285,151.490
C01274=1103.726,128.121,-61.348,177.705,14.286,151.491
C01275=1103.720,127.849,-61.327,177.701,14.287,151.492
C01276=1103.713,127.576,-61.305,177.697,14.287,151.493
C01277=1103.707,127.327,-61.285,177.694,14.288,151.493
C01278=1103.701,127.078,-61.266,177.691,14.289,151.494
C01279=1103.696,126.829,-61.246,177.687,14.289,151.495
C01280=1103.690,126.579,-61.226,177.684,14.290,151.496
C01281=1103.684,126.331,-61.206,177.680,14.290,151.497
C01282=1103.679,126.081,-61.187,177.677,14.291,151.498
C01283=1103.673,125.832,-61.167,177.673,14.291,151.499
C01284=1103.668,125.583,-61.147,177.670,14.292,151.500
C01285=1103.662,125.334,-61.127,177.667,14.292,151.500
C01286=1103.656,125.084,-61.108,177.663,14.293,151.501
C01287=1103.650,124.836,-61.088,177.660,14.293,151.502
C01288=1103.644,124.586,-61.069,177.656,14.293,151.503
C01289=1103.638,124.337,-61.049,177.653,14.294,151.504
C01290=1103.633,124.088,-61.029,177.650,14.295,151.505
C01291=1103.627,123.839,-61.009,177.646,14.295,151.506
C01292=1103.622,123.590,-60.990,177.643,14.296,151.507
C01293=1103.617,123.341,-60.971,177.639,14.296,151.507
C01294=1103.611,123.092,-60.951,177.636,14.297,151.508
C01295=1103.605,122.842,-60.932,177.632,14.297,151.509
C01296=1103.599,122.594,-60.912,177.629,14.298,151.510
C01297=1103.593,122.344,-60.893,177.626,14.299,151.511
C01298=1103.588,122.094,-60.873,177.623,14.298,151.512
C01299=1103.582,121.846,-60.853,177.620,14.299,151.512
C01300=1103.577,121.596,-60.834,177.616,14.300,151.513
C01301=1103.571,121.347,-60.814,177.613,14.300,151.514
C01302=1103.565,121.098,-60.794,177.609,14.300,151.515
C01303=1103.560,120.849,-60.775,177.606,14.301,151.516
C01304=1103.554,120.600,-60.756,177.603,14.302,151.517
C01305=1103.548,120.351,-60.736,177.599,14.302,151.518
C01306=1103.543,120.102,-60.717,177.596,14.303,151.518
C01307=1103.537,119.852,-60.698,177.592,14.302,151.519
C01308=1103.531,119.603,-60.679,177.589,14.303,151.520
C01309=1103.525,119.354,-60.659,177.586,14.304,151.521
C01310=1103.520,119.105,-60.640,177.583,14.304,151.522
C01311=1103.514,118.856,-60.620,177.580,14.305,151.523
C01312=1103.509,118.606,-60.601,177.576,14.305,151.523
C01313=1103.503,118.357,-60.581,177.573,14.305,151.524
C01314=1103.497,118.108,-60.562,177.569,14.306,151.525
C01315=1103.491,117.859,-60.543,177.566,14.306,151.526
C01316=1103.486,117.610,-60.524,177.563,14.307,151.527
C01317=1103.481,117.360,-60.505,177.559,14.307,151.528
C01318=1103.475,117.111,-60.485,177.557,14.307,151.528
C01319=1103.469,116.862,-60.465,177.553,14.308,151.529
C01320=1103.463,116.613,-60.446,177.550,14.308,151.530
C01321=1103.458,116.364,-60.427,177.546,14.308,151.531
C01322=1103.452,116.115,-60.408,177.543,14.309,151.532
C01323=1103.447,115.865,-60.389,177.540,14.310,151.532
C01324=1103.441,115.616,-60.370,177.537,14.309,151.533
C01325=1103.436,115.367,-60.351,177.533,14.310,151.534
C01326=1103.430,115.118,-60.331,177.530,14.310,151.535
C01327=1103.425,114.868,-60.312,177.527,14.311,151.536
C01328=1103.419,114.619,-60.293,177.524,14.312,151.536
C01329=1103.413,114.371,-60.273,177.520,14.312,151.537
C01330=1103.408,114.121,-60.254,177.517,14.312,151.538
C01331=1103.402,113.872,-60.235,177.513,14.312,151.539
C01332=1103.396,113.622,-60.216,177.511,14.313,151.540
C01333=1103.391,113.374,-60.197,177.507,14.313,151.540
C01334=1103.385,113.124,-60.178,177.504,14.314,151.541
C01335=1103.379,112.875,-60.159,177.501,14.314,151.542
C01336=1103.374,112.626,-60.140,177.497,14.314,151.543
C01337=1103.368,112.353,-60.119,177.494,14.315,151.544
C01338=1103.361,112.081,-60.098,177.491,14.315,151.545
C01339=1103.355,111.809,-60.078,177.487,14.315,151.545
C01340=1103.349,111.536,-60.057,177.484,14.316,151.546
C01341=1103.344,111.287,-60.038,177.480,14.316,151.547
C01342=1103.337,111.038,-60.019,177.477,14.316,151.548
C01343=1103.332,110.789,-60.000,177.473,14.317,151.549
C01344=1103.326,110.540,-59.981,177.470,14.317,151.550
C01345=1103.320,110.291,-59.963,177.467,14.318,151.550
C01346=1103.314,110.041,-59.943,177.464,14.318,151.551
C01347=1103.309,109.792,-59.924,177.461,14.319,151.552
C01348=1103.303,109.543,-59.906,177.457,14.318,151.553
C01349=1103.297,109.293,-59.887,177.454,14.319,151.554
C01350=1103.292,109.044,-59.868,177.451,14.319,151.554
C01351=1103.286,108.795,-59.850,177.448,14.319,151.555
C01352=1103.280,108.546,-59.830,177.445,14.320,151.556
C01353=1103.274,108.296,-59.811,177.441,14.320,151.557
C01354=1103.269,108.048,-59.793,177.438,14.321,151.557
C01355=1103.263,107.798,-59.774,177.435,14.321,151.558
C01356=1103.258,107.549,-59.755,177.432,14.321,151.559
C01357=1103.252,107.300,-59.737,177.429,14.321,151.560
C01358=1103.246,107.051,-59.718,177.425,14.321,151.560
C01359=1103.241,106.801,-59.699,177.423,14.322,151.561
C01360=1103.235,106.552,-59.681,177.419,14.323,151.562
C01361=1103.229,106.303,-59.662,177.416,14.323,151.563
C01362=1103.223,106.054,-59.643,177.413,14.323,151.564
C01363=1103.218,105.804,-59.625,177.409,14.323,151.564
C01364=1103.212,105.555,-59.606,177.406,14.324,151.565
C01365=1103.206,105.306,-59.587,177.404,14.324,151.566
C01366=1103.201,105.056,-59.569,177.400,14.324,151.567
C01367=1103.195,104.807,-59.550,177.397,14.324,151.567
C01368=1103.190,104.559,-59.531,177.394,14.324,151.568
C01369=1103.184,104.309,-59.513,177.391,14.325,151.569
C01370=1103.178,104.059,-59.494,177.388,14.325,151.570
C01371=1103.173,103.811,-59.475,177.384,14.325,151.570
C01372=1103.167,103.561,-59.457,177.381,14.326,151.571
C01373=1103.161,103.312,-59.438,177.378,14.326,151.572
C01374=1103.155,103.063,-59.420,177.375,14.326,151.573
C01375=1103.150,102.814,-59.402,177.372,14.327,151.573
C01376=1103.145,102.564,-59.382,177.369,14.326,151.574
C01377=1103.138,102.315,-59.364,177.366,14.327,151.575
C01378=1103.133,102.066,-59.345,177.362,14.327,151.576
C01379=1103.127,101.816,-59.328,177.359,14.327,151.576
C01380=1103.122,101.567,-59.309,177.356,14.328,151.577
C01381=1103.116,101.318,-59.291,177.353,14.327,151.578
C01382=1103.111,101.069,-59.272,177.350,14.328,151.579
C01383=1103.105,100.820,-59.253,177.347,14.328,151.579
C01384=1103.098,100.570,-59.235,177.344,14.328,151.580
C01385=1103.093,100.321,-59.216,177.341,14.329,151.581
C01386=1103.087,100.072,-59.198,177.337,14.329,151.582
C01387=1103.082,99.823,-59.180,177.335,14.329,151.582
C01388=1103.076,99.573,-59.162,177.332,14.330,151.583
C01389=1103.070,99.325,-59.143,177.328,14.330,151.584
C01390=1103.065,99.075,-59.125,177.325,14.330,151.585
C01391=1103.059,98.825,-59.107,177.322,14.330,151.585
C01392=1103.053,98.576,-59.089,177.319,14.330,151.586
C01393=1103.047,98.326,-59.070,177.316,14.331,151.587
C01394=1103.042,98.078,-59.052,177.313,14.330,151.587
C01395=1103.036,97.828,-59.033,177.310,14.331,151.588
C01396=1103.031,97.579,-59.016,177.306,14.331,151.589
C01397=1103.024,97.330,-58.997,177.304,14.331,151.590
C01398=1103.020,97.080,-58.979,177.301,14.332,151.590
C01399=1103.013,96.831,-58.960,177.297,14.331,151.591
C01400=1103.008,96.582,-58.943,177.295,14.332,151.592
C01401=1103.001,96.310,-58.923,177.291,14.332,151.593
C01402=1102.995,96.037,-58.902,177.288,14.332,151.593
C01403=1102.989,95.765,-58.883,177.284,14.333,151.594
C01404=1102.983,95.493,-58.863,177.281,14.332,151.595
C01405=1102.977,95.243,-58.845,177.278,14.332,151.596
C01406=1102.971,94.995,-58.827,177.275,14.333,151.596
C01407=1102.966,94.745,-58.809,177.272,14.333,151.597
C01408=1102.960,94.496,-58.791,177.269,14.333,151.598
C01409=1102.954,94.247,-58.772,177.266,14.333,151.598
C01410=1102.949,93.997,-58.754,177.263,14.333,151.599
C01411=1102.943,93.748,-58.737,177.260,14.334,151.600
C01412=1102.937,93.499,-58.719,177.257,14.333,151.601
C01413=1102.932,93.250,-58.700,177.254,14.334,151.601
C01414=1102.926,93.000,-58.682,177.251,14.334,151.602
C01415=1102.921,92.751,-58.664,177.248,14.334,151.603
C01416=1102.914,92.501,-58.646,177.245,14.334,151.603
C01417=1102.909,92.252,-58.629,177.241,14.334,151.604
C01418=1102.904,92.004,-58.610,177.239,14.334,151.605
C01419=1102.898,91.754,-58.592,177.236,14.335,151.606
C01420=1102.892,91.505,-58.574,177.233,14.334,151.606
C01421=1102.886,91.255,-58.556,177.230,14.335,151.607
C01422=1102.881,91.006,-58.538,177.227,14.335,151.608
C01423=1102.876,90.757,-58.521,177.224,14.335,151.608
C01424=1102.870,90.507,-58.503,177.221,14.335,151.609
C01425=1102.864,90.259,-58.485,177.217,14.335,151.610
C01426=1102.858,90.009,-58.467,177.215,14.335,151.610
C01427=1102.852,89.760,-58.449,177.212,14.336,151.611
C01428=1102.847,89.511,-58.431,177.209,14.335,151.612
C01429=1102.841,89.261,-58.414,177.206,14.336,151.612
C01430=1102.835,89.012,-58.396,177.203,14.336,151.613
C01431=1102.829,88.762,-58.378,177.200,14.336,151.614
C01432=1102.823,88.513,-58.360,177.197,14.336,151.615
C01433=1102.817,88.263,-58.343,177.193,14.336,151.615
C01434=1102.812,88.014,-58.325,177.191,14.336,151.616
C01435=1102.806,87.765,-58.307,177.188,14.336,151.616
C01436=1102.800,87.516,-58.289,177.184,14.336,151.617
C01437=1102.795,87.267,-58.272,177.182,14.337,151.618
C01438=1102.790,87.017,-58.254,177.179,14.337,151.619
C01439=1102.784,86.767,-58.236,177.176,14.337,151.619
C01440=1102.778,86.518,-58.218,177.173,14.337,151.620
C01441=1102.773,86.269,-58.201,177.170,14.337,151.621
C01442=1102.767,86.020,-58.183,177.167,14.337,151.621
C01443=1102.761,85.771,-58.165,177.164,14.337,151.622
C01444=1102.756,85.522,-58.148,177.161,14.337,151.623
C01445=1102.749,85.272,-58.130,177.158,14.337,151.623
C01446=1102.744,85.023,-58.112,177.155,14.337,151.624
C01447=1102.738,84.774,-58.095,177.152,14.337,151.625
C01448=1102.732,84.524,-58.077,177.149,14.337,151.625
C01449=1102.727,84.275,-58.059,177.147,14.337,151.626
C01450=1102.721,84.026,-58.043,177.143,14.337,151.627
C01451=1102.715,83.776,-58.025,177.141,14.337,151.627
C01452=1102.709,83.527,-58.007,177.137,14.337,151.628
C01453=1102.704,83.278,-57.990,177.135,14.337,151.629
C01454=1102.698,83.029,-57.972,177.132,14.338,151.629
C01455=1102.692,82.779,-57.954,177.128,14.337,151.630
C01456=1102.686,82.530,-57.937,177.126,14.338,151.631
C01457=1102.681,82.280,-57.920,177.123,14.338,151.631
C01458=1102.675,82.031,-57.902,177.120,14.338,151.632
C01459=1102.670,81.782,-57.884,177.117,14.338,151.632
C01460=1102.664,81.532,-57.867,177.115,14.338,151.633
C01461=1102.659,81.283,-57.850,177.111,14.338,151.634
C01462=1102.653,81.033,-57.832,177.109,14.338,151.634
C01463=1102.647,80.784,-57.814,177.105,14.337,151.635
C01464=1102.642,80.535,-57.797,177.103,14.338,151.636
C01465=1102.636,80.263,-57.779,177.100,14.338,151.636
C01466=1102.629,79.990,-57.759,177.096,14.338,151.637
C01467=1102.623,79.719,-57.740,177.093,14.337,151.638
C01468=1102.617,79.446,-57.722,177.090,14.338,151.638
C01469=1102.611,79.197,-57.704,177.087,14.337,151.639
C01470=1102.605,78.948,-57.686,177.085,14.337,151.640
C01471=1102.600,78.699,-57.669,177.082,14.338,151.640
C01472=1102.595,78.449,-57.652,177.078,14.337,151.641
C01473=1102.588,78.200,-57.635,177.076,14.337,151.642
C01474=1102.582,77.950,-57.617,177.073,14.337,151.642
C01475=1102.577,77.701,-57.600,177.070,14.337,151.643
C01476=1102.572,77.452,-57.583,177.067,14.337,151.644
C01477=1102.566,77.202,-57.566,177.065,14.337,151.644
C01478=1102.560,76.953,-57.549,177.061,14.337,151.645
C01479=1102.554,76.704,-57.531,177.059,14.337,151.645
C01480=1102.549,76.454,-57.514,177.056,14.338,151.646
C01481=1102.543,76.205,-57.497,177.053,14.337,151.647
C01482=1102.537,75.956,-57.480,177.050,14.337,151.647
C01483=1102.531,75.706,-57.462,177.048,14.337,151.648
C01484=1102.526,75.457,-57.445,177.044,14.337,151.649
C01485=1102.520,75.207,-57.429,177.042,14.337,151.649
C01486=1102.514,74.958,-57.411,177.038,14.337,151.650
C01487=1102.509,74.709,-57.394,177.036,14.337,151.650
C01488=1102.503,74.460,-57.377,177.033,14.337,151.651
C01489=1102.497,74.210,-57.360,177.030,14.336,151.652
C01490=1102.491,73.961,-57.342,177.027,14.337,151.652
C01491=1102.486,73.711,-57.326,177.025,14.337,151.653
C01492=1102.480,73.462,-57.309,177.021,14.336,151.654
C01493=1102.475,73.213,-57.292,177.019,14.337,151.654
C01494=1102.469,72.964,-57.275,177.016,14.337,151.655
C01495=1102.463,72.714,-57.258,177.013,14.336,151.655
C01496=1102.457,72.464,-57.240,177.011,14.336,151.656
C01497=1102.451,72.215,-57.224,177.008,14.336,151.656
C01498=1102.446,71.966,-57.206,177.005,14.336,151.657
C01499=1102.441,71.716,-57.189,177.002,14.336,151.658
C01500=1102.435,71.467,-57.173,177.000,14.336,151.658
C01501=1102.429,71.218,-57.155,176.996,14.336,151.659
C01502=1102.423,70.969,-57.139,176.994,14.336,151.660
C01503=1102.418,70.720,-57.122,176.991,14.336,151.660
C01504=1102.412,70.470,-57.105,176.988,14.336,151.661
C01505=1102.406,70.221,-57.089,176.985,14.336,151.661
C01506=1102.401,69.972,-57.071,176.983,14.336,151.662
C01507=1102.394,69.721,-57.054,176.980,14.335,151.663
C01508=1102.389,69.472,-57.037,176.977,14.335,151.663
C01509=1102.383,69.223,-57.021,176.975,14.335,151.664
C01510=1102.378,68.973,-57.004,176.971,14.335,151.664
C01511=1102.372,68.724,-56.987,176.969,14.335,151.665
C01512=1102.366,68.475,-56.970,176.966,14.335,151.665
C01513=1102.360,68.226,-56.954,176.963,14.335,151.666
C01514=1102.355,67.976,-56.937,176.960,14.335,151.667
C01515=1102.349,67.727,-56.920,176.958,14.335,151.667
C01516=1102.344,67.478,-56.903,176.955,14.334,151.668
C01517=1102.338,67.228,-56.887,176.952,14.334,151.668
C01518=1102.332,66.979,-56.870,176.950,14.334,151.669
C01519=1102.326,66.730,-56.853,176.946,14.334,151.670
C01520=1102.321,66.480,-56.836,176.944,14.334,151.670
C01521=1102.314,66.230,-56.819,176.942,14.334,151.671
C01522=1102.309,65.981,-56.803,176.938,14.333,151.671
C01523=1102.303,65.731,-56.786,176.936,14.333,151.672
C01524=1102.298,65.482,-56.769,176.933,14.333,151.672
C01525=1102.292,65.233,-56.752,176.930,14.333,151.673
C01526=1102.286,64.983,-56.736,176.928,14.333,151.674
C01527=1102.281,64.734,-56.719,176.925,14.333,151.674
C01528=1102.275,64.484,-56.703,176.922,14.332,151.675
C01529=1102.268,64.212,-56.685,176.919,14.333,151.675
C01530=1102.262,63.940,-56.667,176.916,14.332,151.676
C01531=1102.256,63.669,-56.648,176.913,14.332,151.677
C01532=1102.249,63.397,-56.631,176.910,14.332,151.677
C01533=1102.244,63.146,-56.613,176.907,14.332,151.678
C01534=1102.238,62.897,-56.597,176.905,14.332,151.678
C01535=1102.232,62.647,-56.581,176.902,14.331,151.679
C01536=1102.226,62.398,-56.565,176.899,14.331,151.680
C01537=1102.221,62.148,-56.548,176.897,14.331,151.680
C01538=1102.215,61.899,-56.531,176.894,14.331,151.681
C01539=1102.209,61.650,-56.515,176.891,14.331,151.681
C01540=1102.203,61.400,-56.499,176.889,14.331,151.682
C01541=1102.197,61.151,-56.482,176.885,14.331,151.683
C01542=1102.192,60.901,-56.466,176.883,14.330,151.683
C01543=1102.185,60.653,-56.449,176.881,14.330,151.684
C01544=1102.179,60.403,-56.433,176.878,14.330,151.684
C01545=1102.174,60.154,-56.416,176.875,14.330,151.685
C01546=1102.168,59.904,-56.399,176.872,14.330,151.685
C01547=1102.162,59.655,-56.383,176.870,14.330,151.686
C01548=1102.156,59.406,-56.367,176.867,14.329,151.686
C01549=1102.151,59.156,-56.350,176.864,14.329,151.687
C01550=1102.146,58.907,-56.334,176.862,14.329,151.688
C01551=1102.140,58.657,-56.319,176.858,14.329,151.688
C01552=1102.134,58.408,-56.302,176.856,14.329,151.689
C01553=1102.128,58.159,-56.286,176.854,14.329,151.689
C01554=1102.123,57.909,-56.269,176.850,14.328,151.690
C01555=1102.117,57.660,-56.253,176.848,14.328,151.690
C01556=1102.111,57.410,-56.237,176.846,14.328,151.691
C01557=1102.105,57.161,-56.221,176.843,14.328,151.691
C01558=1102.099,56.912,-56.204,176.840,14.327,151.692
C01559=1102.093,56.662,-56.188,176.838,14.327,151.692
C01560=1102.088,56.413,-56.171,176.835,14.327,151.693
C01561=1102.082,56.163,-56.155,176.832,14.327,151.694
C01562=1102.076,55.913,-56.139,176.829,14.327,151.694
C01563=1102.071,55.665,-56.124,176.827,14.326,151.695
C01564=1102.065,55.415,-56.107,176.824,14.326,151.695
C01565=1102.059,55.166,-56.091,176.821,14.326,151.696
C01566=1102.053,54.917,-56.075,176.819,14.326,151.696
C01567=1102.048,54.667,-56.058,176.817,14.326,151.697
C01568=1102.042,54.417,-56.042,176.814,14.325,151.697
C01569=1102.036,54.168,-56.026,176.811,14.325,151.698
C01570=1102.030,53.918,-56.010,176.809,14.325,151.698
C01571=1102.025,53.670,-55.994,176.806,14.324,151.699
C01572=1102.019,53.420,-55.978,176.803,14.324,151.699
C01573=1102.013,53.170,-55.962,176.801,14.324,151.700
C01574=1102.007,52.921,-55.946,176.799,14.324,151.700
C01575=1102.002,52.672,-55.930,176.795,14.323,151.701
C01576=1101.996,52.422,-55.913,176.793,14.323,151.701
C01577=1101.991,52.173,-55.898,176.791,14.323,151.702
C01578=1101.985,51.923,-55.881,176.788,14.322,151.702
C01579=1101.979,51.674,-55.865,176.785,14.322,151.703
C01580=1101.974,51.424,-55.850,176.783,14.322,151.704
C01581=1101.968,51.175,-55.833,176.780,14.321,151.704
C01582=1101.962,50.926,-55.817,176.777,14.322,151.705
C01583=1101.956,50.677,-55.801,176.775,14.321,151.705
C01584=1101.951,50.427,-55.786,176.772,14.321,151.706
C01585=1101.945,50.177,-55.769,176.769,14.320,151.706
C01586=1101.939,49.928,-55.753,176.767,14.321,151.707
C01587=1101.934,49.679,-55.738,176.765,14.320,151.707
C01588=1101.928,49.429,-55.722,176.762,14.320,151.708
C01589=1101.922,49.179,-55.706,176.759,14.319,151.708
C01590=1101.916,48.930,-55.690,176.757,14.319,151.709
C01591=1101.911,48.681,-55.674,176.755,14.319,151.709
C01592=1101.905,48.431,-55.658,176.751,14.319,151.710
C01593=1101.899,48.159,-55.640,176.749,14.318,151.710
C01594=1101.893,47.887,-55.623,176.746,14.318,151.711
C01595=1101.887,47.614,-55.606,176.743,14.318,151.711
C01596=1101.881,47.341,-55.589,176.740,14.317,151.712
C01597=1101.875,47.092,-55.573,176.738,14.317,151.712
C01598=1101.869,46.843,-55.557,176.736,14.317,151.713
C01599=1101.864,46.593,-55.542,176.732,14.316,151.713
C01600=1101.858,46.344,-55.525,176.730,14.316,151.714
C01601=1101.852,46.094,-55.510,176.728,14.315,151.714
C01602=1101.847,45.845,-55.494,176.725,14.316,151.715
C01603=1101.841,45.595,-55.478,176.723,14.315,151.715
C01604=1101.835,45.346,-55.462,176.720,14.315,151.716
C01605=1101.830,45.096,-55.447,176.718,14.314,151.716
C01606=1101.824,44.847,-55.431,176.716,14.314,151.717
C01607=1101.819,44.598,-55.415,176.712,14.314,151.717
C01608=1101.813,44.348,-55.400,176.710,14.313,151.718
C01609=1101.808,44.099,-55.384,176.708,14.313,151.718
C01610=1101.802,43.849,-55.368,176.705,14.312,151.719
C01611=1101.796,43.600,-55.352,176.703,14.312,151.719
C01612=1101.791,43.350,-55.337,176.700,14.312,151.720
C01613=1101.784,43.101,-55.321,176.698,14.312,151.720
C01614=1101.779,42.851,-55.306,176.695,14.311,151.721
C01615=1101.774,42.602,-55.290,176.692,14.311,151.721
C01616=1101.768,42.353,-55.274,176.690,14.311,151.722
C01617=1101.762,42.103,-55.259,176.688,14.310,151.722
C01618=1101.756,41.854,-55.244,176.685,14.310,151.723
C01619=1101.750,41.604,-55.228,176.682,14.309,151.723
C01620=1101.745,41.354,-55.212,176.680,14.309,151.724
C01621=1101.739,41.106,-55.196,176.678,14.309,151.724
C01622=1101.734,40.856,-55.181,176.675,14.308,151.725
C01623=1101.727,40.606,-55.166,176.673,14.308,151.725
C01624=1101.722,40.358,-55.150,176.670,14.308,151.726
C01625=1101.716,40.108,-55.134,176.667,14.307,151.726
C01626=1101.711,39.858,-55.119,176.665,14.307,151.726
C01627=1101.705,39.609,-55.104,176.662,14.307,151.727
C01628=1101.699,39.359,-55.088,176.660,14.306,151.727
C01629=1101.693,39.109,-55.073,176.657,14.306,151.728
C01630=1101.688,38.860,-55.057,176.655,14.305,151.728
C01631=1101.681,38.611,-55.042,176.653,14.305,151.729
C01632=1101.676,38.361,-55.026,176.650,14.305,151.729
C01633=1101.671,38.112,-55.011,176.647,14.304,151.730
C01634=1101.665,37.862,-54.995,176.645,14.304,151.730
C01635=1101.659,37.614,-54.980,176.643,14.304,151.731
C01636=1101.653,37.364,-54.965,176.641,14.303,151.731
C01637=1101.647,37.114,-54.950,176.638,14.302,151.732
C01638=1101.642,36.865,-54.935,176.635,14.303,151.732
C01639=1101.636,36.615,-54.919,176.633,14.302,151.733
C01640=1101.630,36.366,-54.903,176.631,14.302,151.733
C01641=1101.625,36.116,-54.888,176.628,14.301,151.734
C01642=1101.618,35.867,-54.873,176.625,14.301,151.734
C01643=1101.613,35.617,-54.858,176.623,14.301,151.735
C01644=1101.607,35.367,-54.842,176.621,14.300,151.735
C01645=1101.601,35.118,-54.828,176.619,14.300,151.735
C01646=1101.596,34.869,-54.812,176.615,14.300,151.736
C01647=1101.589,34.620,-54.797,176.613,14.299,151.736
C01648=1101.584,34.370,-54.782,176.611,14.299,151.737
C01649=1101.578,34.121,-54.767,176.609,14.299,151.737
C01650=1101.572,33.871,-54.751,176.606,14.298,151.738
C01651=1101.567,33.621,-54.736,176.603,14.298,151.738
C01652=1101.561,33.372,-54.721,176.601,14.297,151.739
C01653=1101.556,33.122,-54.706,176.599,14.297,151.739
C01654=1101.549,32.873,-54.691,176.596,14.296,151.740
C01655=1101.544,32.624,-54.675,176.594,14.296,151.740
C01656=1101.538,32.374,-54.660,176.592,14.295,151.740
C01657=1101.532,32.101,-54.643,176.588,14.295,151.741
C01658=1101.526,31.829,-54.627,176.586,14.295,151.742
C01659=1101.519,31.557,-54.611,176.584,14.294,151.742
C01660=1101.513,31.284,-54.594,176.581,14.294,151.743
C01661=1101.508,31.035,-54.579,176.578,14.293,151.743
C01662=1101.501,30.786,-54.564,176.576,14.293,151.743
C01663=1101.496,30.536,-54.549,176.573,14.292,151.744
C01664=1101.490,30.287,-54.534,176.571,14.292,151.744
C01665=1101.485,30.037,-54.518,176.569,14.291,151.745
C01666=1101.478,29.788,-54.504,176.567,14.291,151.745
C01667=1101.473,29.538,-54.488,176.564,14.291,151.746
C01668=1101.467,29.288,-54.474,176.561,14.290,151.746
C01669=1101.462,29.039,-54.459,176.559,14.290,151.747
C01670=1101.456,28.789,-54.444,176.557,14.290,151.747
C01671=1101.451,28.540,-54.429,176.555,14.289,151.747
C01672=1101.444,28.290,-54.414,176.552,14.289,151.748
C01673=1101.438,28.041,-54.399,176.550,14.288,151.748
C01674=1101.433,27.791,-54.384,176.547,14.288,151.749
C01675=1101.427,27.542,-54.369,176.545,14.287,151.749
C01676=1101.422,27.292,-54.354,176.543,14.287,151.750
C01677=1101.415,27.043,-54.339,176.540,14.286,151.750
C01678=1101.409,26.794,-54.324,176.538,14.286,151.750
C01679=1101.405,26.544,-54.310,176.535,14.286,151.751
C01680=1101.398,26.294,-54.295,176.533,14.286,151.751
C01681=1101.393,26.045,-54.280,176.531,14.285,151.752
C01682=1101.387,25.795,-54.265,176.528,14.284,151.752
C01683=1101.381,25.546,-54.250,176.526,14.284,151.753
C01684=1101.375,25.297,-54.235,176.524,14.284,151.753
C01685=1101.370,25.048,-54.220,176.521,14.283,151.754
C01686=1101.364,24.797,-54.206,176.519,14.283,151.754
C01687=1101.358,24.548,-54.191,176.516,14.282,151.754
C01688=1101.352,24.298,-54.176,176.514,14.282,151.755
C01689=1101.346,24.049,-54.161,176.512,14.281,151.755
C01690=1101.340,23.800,-54.146,176.510,14.281,151.756
C01691=1101.335,23.550,-54.132,176.507,14.281,151.756
C01692=1101.329,23.300,-54.117,176.504,14.280,151.757
C01693=1101.323,23.051,-54.102,176.502,14.279,151.757
C01694=1101.317,22.802,-54.087,176.500,14.279,151.757
C01695=1101.312,22.552,-54.073,176.498,14.279,151.758
C01696=1101.306,22.303,-54.058,176.496,14.278,151.758
C01697=1101.300,22.053,-54.043,176.493,14.277,151.759
C01698=1101.294,21.803,-54.029,176.491,14.277,151.759
C01699=1101.289,21.554,-54.014,176.488,14.277,151.760
C01700=1101.283,21.305,-53.999,176.486,14.276,151.760
C01701=1101.277,21.056,-53.985,176.484,14.276,151.760
C01702=1101.271,20.805,-53.970,176.481,14.275,151.761
C01703=1101.266,20.556,-53.955,176.479,14.275,151.761
C01704=1101.260,20.307,-53.941,176.477,14.274,151.762
C01705=1101.254,20.057,-53.926,176.475,14.274,151.762
C01706=1101.248,19.808,-53.912,176.473,14.273,151.762
C01707=1101.242,19.558,-53.897,176.470,14.272,151.763
C01708=1101.237,19.308,-53.882,176.467,14.272,151.763
C01709=1101.231,19.059,-53.868,176.465,14.272,151.764
C01710=1101.225,18.809,-53.854,176.463,14.272,151.764
C01711=1101.220,18.560,-53.839,176.461,14.271,151.765
C01712=1101.213,18.310,-53.824,176.459,14.271,151.765
C01713=1101.208,18.061,-53.810,176.456,14.270,151.765
C01714=1101.203,17.812,-53.795,176.454,14.270,151.766
C01715=1101.197,17.561,-53.781,176.451,14.269,151.766
C01716=1101.191,17.312,-53.766,176.449,14.269,151.767
C01717=1101.185,17.063,-53.752,176.447,14.268,151.767
C01718=1101.179,16.813,-53.737,176.445,14.268,151.767
C01719=1101.173,16.564,-53.723,176.442,14.267,151.768
C01720=1101.168,16.315,-53.709,176.440,14.267,151.768
C01721=1101.162,16.043,-53.693,176.438,14.266,151.769
C01722=1101.155,15.772,-53.677,176.435,14.265,151.769
C01723=1101.149,15.501,-53.662,176.433,14.265,151.770
C01724=1101.142,15.230,-53.646,176.430,14.265,151.770
C01725=1101.137,14.981,-53.631,176.428,14.264,151.770
C01726=1101.131,14.731,-53.617,176.425,14.263,151.771
C01727=1101.126,14.482,-53.602,176.423,14.263,151.771
C01728=1101.120,14.232,-53.588,176.421,14.263,151.772
C01729=1101.114,13.982,-53.574,176.419,14.262,151.772
C01730=1101.108,13.733,-53.560,176.417,14.262,151.772
C01731=1101.102,13.484,-53.545,176.415,14.261,151.773
C01732=1101.096,13.234,-53.531,176.412,14.260,151.773
C01733=1101.091,12.984,-53.517,176.409,14.260,151.774
C01734=1101.085,12.735,-53.502,176.407,14.260,151.774
C01735=1101.078,12.485,-53.489,176.405,14.259,151.774
C01736=1101.073,12.236,-53.474,176.403,14.259,151.775
C01737=1101.067,11.987,-53.460,176.401,14.259,151.775
C01738=1101.061,11.737,-53.445,176.398,14.257,151.776
C01739=1101.055,11.487,-53.431,176.396,14.257,151.776
C01740=1101.050,11.238,-53.418,176.394,14.257,151.776
C01741=1101.043,10.988,-53.403,176.391,14.256,151.777
C01742=1101.038,10.738,-53.389,176.389,14.256,151.777
C01743=1101.032,10.489,-53.375,176.387,14.256,151.778
C01744=1101.027,10.240,-53.360,176.385,14.255,151.778
C01745=1101.021,9.990,-53.346,176.382,14.254,151.778
C01746=1101.015,9.740,-53.332,176.380,14.254,151.779
C01747=1101.009,9.491,-53.318,176.378,14.253,151.779
C01748=1101.002,9.241,-53.304,176.376,14.253,151.780
C01749=1100.997,8.992,-53.290,176.374,14.252,151.780
C01750=1100.991,8.743,-53.276,176.372,14.252,151.780
C01751=1100.986,8.493,-53.262,176.369,14.252,151.781
C01752=1100.980,8.243,-53.248,176.366,14.251,151.781
C01753=1100.974,7.994,-53.233,176.365,14.250,151.782
C01754=1100.968,7.744,-53.219,176.362,14.249,151.782
C01755=1100.963,7.495,-53.205,176.360,14.249,151.782
C01756=1100.956,7.245,-53.192,176.358,14.249,151.783
C01757=1100.950,6.996,-53.177,176.356,14.249,151.783
C01758=1100.945,6.746,-53.163,176.354,14.248,151.783
C01759=1100.939,6.497,-53.149,176.351,14.247,151.784
C01760=1100.933,6.246,-53.135,176.349,14.246,151.784
C01761=1100.928,5.997,-53.121,176.347,14.246,151.785
C01762=1100.921,5.748,-53.107,176.345,14.245,151.785
C01763=1100.916,5.499,-53.093,176.343,14.245,151.785
C01764=1100.910,5.249,-53.079,176.340,14.245,151.786
C01765=1100.904,4.999,-53.065,176.338,14.244,151.786
C01766=1100.899,4.749,-53.051,176.336,14.244,151.787
C01767=1100.893,4.500,-53.037,176.333,14.243,151.787
C01768=1100.887,4.251,-53.024,176.331,14.242,151.787
C01769=1100.881,4.001,-53.010,176.329,14.242,151.788
C01770=1100.876,3.752,-52.996,176.327,14.241,151.788
C01771=1100.870,3.501,-52.982,176.325,14.241,151.789
C01772=1100.864,3.252,-52.968,176.323,14.240,151.789
C01773=1100.858,3.003,-52.954,176.321,14.240,151.789
C01774=1100.853,2.753,-52.941,176.319,14.240,151.790
C01775=1100.847,2.504,-52.926,176.316,14.238,151.790
C01776=1100.841,2.255,-52.912,176.314,14.238,151.790
C01777=1100.835,2.005,-52.898,176.312,14.237,151.791
C01778=1100.829,1.755,-52.885,176.310,14.237,151.791
C01779=1100.824,1.505,-52.871,176.308,14.236,151.791
C01780=1100.818,1.256,-52.857,176.305,14.236,151.792
C01781=1100.813,1.006,-52.843,176.303,14.235,151.792
C01782=1100.806,0.757,-52.830,176.301,14.235,151.793
C01783=1100.801,0.507,-52.816,176.298,14.234,151.793
C01784=1100.795,0.258,-52.802,176.296,14.233,151.793
C01785=1100.789,-0.011,-52.787,176.294,14.233,151.794
C01786=1100.782,-0.281,-52.773,176.292,14.233,151.794
C01787=1100.776,-0.549,-52.758,176.289,14.232,151.795
C01788=1100.771,-0.819,-52.742,176.287,14.231,151.795
C01789=1100.764,-1.068,-52.729,176.285,14.231,151.795
C01790=1100.759,-1.317,-52.715,176.283,14.230,151.796
C01791=1100.753,-1.567,-52.701,176.281,14.229,151.796
C01792=1100.748,-1.817,-52.687,176.279,14.229,151.796
C01793=1100.742,-2.066,-52.674,176.277,14.228,151.797
C01794=1100.736,-2.316,-52.660,176.275,14.228,151.797
C01795=1100.730,-2.566,-52.646,176.272,14.227,151.797
C01796=1100.724,-2.816,-52.633,176.270,14.226,151.798
C01797=1100.719,-3.065,-52.620,176.268,14.226,151.798
C01798=1100.713,-3.315,-52.606,176.266,14.225,151.799
C01799=1100.707,-3.564,-52.592,176.264,14.225,151.799
C01800=1100.702,-3.814,-52.579,176.262,14.224,151.799
C01801=1100.695,-4.063,-52.565,176.260,14.224,151.800
C01802=1100.690,-4.312,-52.551,176.257,14.223,151.800
C01803=1100.684,-4.562,-52.538,176.256,14.223,151.800
C01804=1100.678,-4.811,-52.524,176.253,14.222,151.801
